C09080=1091.233,-110.223,-49.572,174.703,15.869,152.459
C09081=1091.239,-109.973,-49.581,174.704,15.869,152.459
C09082=1091.245,-109.724,-49.590,174.706,15.870,152.459
C09083=1091.251,-109.474,-49.600,174.708,15.871,152.459
C09084=1091.257,-109.224,-49.610,174.709,15.871,152.458
C09085=1091.263,-108.974,-49.619,174.711,15.872,152.458
C09086=1091.270,-108.724,-49.629,174.713,15.872,152.458
C09087=1091.275,-108.475,-49.640,174.714,15.872,152.458
C09088=1091.281,-108.225,-49.649,174.716,15.873,152.457
C09089=1091.288,-107.975,-49.659,174.717,15.874,152.457
C09090=1091.294,-107.726,-49.668,174.719,15.874,152.457
C09091=1091.300,-107.476,-49.678,174.720,15.875,152.457
C09092=1091.306,-107.226,-49.687,174.722,15.875,152.457
C09093=1091.312,-106.976,-49.697,174.723,15.875,152.456
C09094=1091.318,-106.727,-49.708,174.725,15.877,152.456
C09095=1091.324,-106.477,-49.717,174.727,15.877,152.456
C09096=1091.330,-106.227,-49.727,174.729,15.878,152.456
C09097=1091.337,-105.977,-49.737,174.730,15.878,152.456
C09098=1091.343,-105.727,-49.746,174.732,15.879,152.455
C09099=1091.349,-105.478,-49.757,174.733,15.880,152.455
C09100=1091.355,-105.228,-49.767,174.735,15.880,152.455
C09101=1091.361,-104.978,-49.776,174.736,15.880,152.455
C09102=1091.367,-104.729,-49.786,174.738,15.881,152.454
C09103=1091.372,-104.478,-49.796,174.739,15.882,152.454
C09104=1091.379,-104.229,-49.806,174.741,15.882,152.454
C09105=1091.385,-103.980,-49.816,174.743,15.883,152.454
C09106=1091.391,-103.730,-49.825,174.745,15.884,152.454
C09107=1091.397,-103.480,-49.835,174.746,15.884,152.453
C09108=1091.403,-103.230,-49.846,174.748,15.885,152.453
C09109=1091.409,-102.981,-49.855,174.750,15.885,152.453
C09110=1091.416,-102.731,-49.865,174.750,15.886,152.453
C09111=1091.422,-102.481,-49.874,174.752,15.887,152.453
C09112=1091.427,-102.232,-49.885,174.754,15.887,152.452
C09113=1091.434,-101.982,-49.895,174.756,15.888,152.452
C09114=1091.440,-101.732,-49.904,174.757,15.889,152.452
C09115=1091.446,-101.482,-49.915,174.759,15.889,152.452
C09116=1091.452,-101.233,-49.925,174.761,15.890,152.451
C09117=1091.458,-100.983,-49.934,174.762,15.890,152.451
C09118=1091.464,-100.733,-49.944,174.763,15.891,152.451
C09119=1091.470,-100.484,-49.955,174.765,15.892,152.451
C09120=1091.476,-100.234,-49.964,174.767,15.892,152.451
C09121=1091.482,-99.984,-49.974,174.768,15.893,152.451
C09122=1091.488,-99.734,-49.985,174.770,15.894,152.450
C09123=1091.495,-99.484,-49.995,174.772,15.894,152.450
C09124=1091.501,-99.234,-50.004,174.773,15.895,152.450
C09125=1091.507,-98.985,-50.015,174.775,15.895,152.450
C09126=1091.513,-98.735,-50.025,174.776,15.896,152.449
C09127=1091.519,-98.486,-50.035,174.778,15.897,152.449
C09128=1091.525,-98.236,-50.045,174.780,15.898,152.449
C09129=1091.531,-97.986,-50.055,174.781,15.898,152.449
C09130=1091.537,-97.737,-50.065,174.783,15.899,152.449
C09131=1091.543,-97.487,-50.075,174.785,15.900,152.448
C09132=1091.550,-97.211,-50.086,174.786,15.900,152.448
C09133=1091.556,-96.936,-50.098,174.788,15.901,152.448
C09134=1091.563,-96.661,-50.109,174.790,15.902,152.448
C09135=1091.570,-96.385,-50.119,174.791,15.902,152.448
C09136=1091.575,-96.135,-50.130,174.793,15.903,152.447
C09137=1091.582,-95.886,-50.140,174.795,15.904,152.447
C09138=1091.587,-95.636,-50.150,174.796,15.905,152.447
C09139=1091.593,-95.387,-50.160,174.798,15.906,152.447
C09140=1091.600,-95.136,-50.171,174.799,15.906,152.447
C09141=1091.606,-94.887,-50.181,174.801,15.907,152.446
C09142=1091.611,-94.637,-50.191,174.803,15.908,152.446
C09143=1091.618,-94.387,-50.201,174.805,15.908,152.446
C09144=1091.623,-94.138,-50.212,174.805,15.909,152.446
C09145=1091.629,-93.888,-50.221,174.807,15.910,152.446
C09146=1091.635,-93.638,-50.232,174.809,15.911,152.446
C09147=1091.641,-93.388,-50.242,174.811,15.911,152.445
C09148=1091.647,-93.139,-50.253,174.812,15.911,152.445
C09149=1091.653,-92.889,-50.262,174.813,15.913,152.445
C09150=1091.659,-92.640,-50.273,174.815,15.913,152.445
C09151=1091.665,-92.390,-50.283,174.817,15.914,152.445
C09152=1091.671,-92.140,-50.294,174.819,15.915,152.444
C09153=1091.678,-91.890,-50.303,174.820,15.916,152.444
C09154=1091.683,-91.640,-50.314,174.822,15.916,152.444
C09155=1091.690,-91.391,-50.324,174.824,15.917,152.444
C09156=1091.695,-91.141,-50.335,174.825,15.918,152.444
C09157=1091.701,-90.892,-50.346,174.826,15.918,152.443
C09158=1091.707,-90.642,-50.355,174.828,15.919,152.443
C09159=1091.713,-90.392,-50.366,174.830,15.920,152.443
C09160=1091.719,-90.143,-50.376,174.831,15.921,152.443
C09161=1091.726,-89.892,-50.387,174.833,15.922,152.443
C09162=1091.732,-89.643,-50.396,174.834,15.922,152.442
C09163=1091.737,-89.393,-50.407,174.836,15.923,152.442
C09164=1091.744,-89.144,-50.418,174.838,15.924,152.442
C09165=1091.749,-88.894,-50.428,174.839,15.925,152.442
C09166=1091.755,-88.644,-50.439,174.841,15.925,152.442
C09167=1091.761,-88.394,-50.448,174.842,15.926,152.442
C09168=1091.768,-88.144,-50.460,174.844,15.927,152.441
C09169=1091.774,-87.895,-50.470,174.846,15.928,152.441
C09170=1091.780,-87.645,-50.480,174.848,15.928,152.441
C09171=1091.786,-87.396,-50.490,174.849,15.930,152.441
C09172=1091.791,-87.146,-50.500,174.850,15.930,152.441
C09173=1091.797,-86.896,-50.511,174.852,15.931,152.441
C09174=1091.804,-86.646,-50.522,174.854,15.931,152.440
C09175=1091.810,-86.396,-50.532,174.856,15.932,152.440
C09176=1091.816,-86.147,-50.542,174.857,15.933,152.440
C09177=1091.822,-85.898,-50.553,174.858,15.933,152.440
C09178=1091.828,-85.648,-50.563,174.860,15.934,152.440
C09179=1091.834,-85.398,-50.574,174.862,15.935,152.439
C09180=1091.840,-85.148,-50.585,174.864,15.936,152.439
C09181=1091.846,-84.898,-50.594,174.865,15.937,152.439
C09182=1091.852,-84.649,-50.605,174.866,15.937,152.439
C09183=1091.858,-84.399,-50.616,174.868,15.938,152.439
C09184=1091.865,-84.149,-50.627,174.870,15.939,152.438
C09185=1091.870,-83.899,-50.637,174.872,15.940,152.438
C09186=1091.877,-83.650,-50.647,174.873,15.941,152.438
C09187=1091.883,-83.401,-50.658,174.875,15.942,152.438
C09188=1091.889,-83.150,-50.669,174.876,15.942,152.438
C09189=1091.895,-82.901,-50.679,174.878,15.943,152.438
C09190=1091.901,-82.651,-50.690,174.879,15.944,152.437
C09191=1091.907,-82.402,-50.701,174.881,15.945,152.437
C09192=1091.914,-82.152,-50.711,174.883,15.946,152.437
C09193=1091.919,-81.902,-50.722,174.885,15.946,152.437
C09194=1091.926,-81.652,-50.732,174.886,15.947,152.437
C09195=1091.931,-81.403,-50.743,174.888,15.948,152.436
C09196=1091.938,-81.130,-50.754,174.889,15.949,152.436
C09197=1091.945,-80.856,-50.766,174.891,15.950,152.436
C09198=1091.951,-80.584,-50.778,174.893,15.951,152.436
C09199=1091.958,-80.310,-50.789,174.895,15.951,152.436
C09200=1091.964,-80.061,-50.800,174.896,15.952,152.436
C09201=1091.970,-79.812,-50.811,174.898,15.953,152.435
C09202=1091.976,-79.561,-50.821,174.900,15.954,152.435
C09203=1091.982,-79.311,-50.832,174.902,15.955,152.435
C09204=1091.988,-79.062,-50.843,174.903,15.956,152.435
C09205=1091.994,-78.812,-50.854,174.904,15.956,152.435
C09206=1092.001,-78.562,-50.864,174.906,15.957,152.435
C09207=1092.006,-78.313,-50.875,174.908,15.958,152.434
C09208=1092.012,-78.063,-50.886,174.909,15.959,152.434
C09209=1092.018,-77.813,-50.896,174.911,15.960,152.434
C09210=1092.024,-77.563,-50.908,174.913,15.961,152.434
C09211=1092.030,-77.314,-50.918,174.915,15.962,152.434
C09212=1092.036,-77.064,-50.929,174.915,15.963,152.434
C09213=1092.042,-76.815,-50.940,174.917,15.963,152.433
C09214=1092.048,-76.565,-50.951,174.919,15.964,152.433
C09215=1092.054,-76.315,-50.962,174.921,15.965,152.433
C09216=1092.060,-76.066,-50.973,174.922,15.966,152.433
C09217=1092.065,-75.816,-50.983,174.924,15.967,152.433
C09218=1092.072,-75.566,-50.993,174.926,15.968,152.433
C09219=1092.078,-75.316,-51.004,174.927,15.969,152.432
C09220=1092.084,-75.067,-51.015,174.929,15.969,152.432
C09221=1092.090,-74.817,-51.026,174.930,15.970,152.432
C09222=1092.096,-74.567,-51.037,174.932,15.972,152.432
C09223=1092.101,-74.318,-51.048,174.934,15.972,152.432
C09224=1092.107,-74.068,-51.059,174.935,15.973,152.432
C09225=1092.114,-73.818,-51.070,174.937,15.974,152.432
C09226=1092.119,-73.568,-51.081,174.939,15.975,152.431
C09227=1092.125,-73.319,-51.092,174.940,15.976,152.431
C09228=1092.131,-73.070,-51.103,174.941,15.977,152.431
C09229=1092.137,-72.819,-51.114,174.943,15.977,152.431
C09230=1092.143,-72.570,-51.125,174.945,15.979,152.431
C09231=1092.149,-72.320,-51.136,174.946,15.980,152.431
C09232=1092.154,-72.071,-51.147,174.948,15.981,152.431
C09233=1092.161,-71.821,-51.158,174.950,15.982,152.430
C09234=1092.166,-71.571,-51.169,174.951,15.983,152.430
C09235=1092.172,-71.322,-51.180,174.953,15.984,152.430
C09236=1092.179,-71.071,-51.191,174.955,15.985,152.430
C09237=1092.184,-70.822,-51.202,174.957,15.986,152.430
C09238=1092.190,-70.572,-51.213,174.957,15.986,152.430
C09239=1092.196,-70.323,-51.224,174.959,15.987,152.429
C09240=1092.202,-70.073,-51.235,174.961,15.988,152.429
C09241=1092.208,-69.823,-51.246,174.962,15.989,152.429
C09242=1092.213,-69.574,-51.257,174.964,15.990,152.429
C09243=1092.219,-69.323,-51.269,174.966,15.991,152.429
C09244=1092.225,-69.074,-51.279,174.968,15.992,152.429
C09245=1092.231,-68.825,-51.291,174.969,15.993,152.429
C09246=1092.237,-68.575,-51.302,174.971,15.994,152.428
C09247=1092.243,-68.325,-51.313,174.973,15.995,152.428
C09248=1092.249,-68.076,-51.324,174.974,15.996,152.428
C09249=1092.254,-67.826,-51.335,174.975,15.997,152.428
C09250=1092.261,-67.576,-51.346,174.977,15.998,152.428
C09251=1092.267,-67.327,-51.357,174.979,15.999,152.428
C09252=1092.272,-67.077,-51.368,174.980,16.000,152.428
C09253=1092.278,-66.827,-51.380,174.982,16.001,152.427
C09254=1092.284,-66.578,-51.391,174.984,16.002,152.427
C09255=1092.290,-66.328,-51.403,174.985,16.003,152.427
C09256=1092.296,-66.078,-51.413,174.987,16.004,152.427
C09257=1092.302,-65.829,-51.424,174.989,16.005,152.427
C09258=1092.308,-65.578,-51.436,174.990,16.006,152.427
C09259=1092.314,-65.329,-51.446,174.992,16.007,152.426
C09260=1092.320,-65.058,-51.459,174.994,16.008,152.426
C09261=1092.327,-64.788,-51.471,174.995,16.009,152.426
C09262=1092.333,-64.517,-51.483,174.997,16.010,152.426
C09263=1092.340,-64.245,-51.495,174.999,16.011,152.426
C09264=1092.345,-63.995,-51.507,175.001,16.012,152.426
C09265=1092.351,-63.746,-51.518,175.002,16.013,152.426
C09266=1092.357,-63.496,-51.530,175.004,16.014,152.425
C09267=1092.363,-63.247,-51.541,175.005,16.015,152.425
C09268=1092.369,-62.997,-51.552,175.007,16.016,152.425
C09269=1092.376,-62.748,-51.563,175.009,16.017,152.425
C09270=1092.381,-62.498,-51.574,175.011,16.018,152.425
C09271=1092.387,-62.248,-51.586,175.012,16.019,152.425
C09272=1092.393,-61.998,-51.597,175.014,16.020,152.424
C09273=1092.399,-61.749,-51.609,175.016,16.021,152.424
C09274=1092.405,-61.499,-51.620,175.017,16.022,152.424
C09275=1092.411,-61.249,-51.631,175.018,16.023,152.424
C09276=1092.417,-61.000,-51.643,175.020,16.023,152.424
C09277=1092.422,-60.750,-51.654,175.022,16.025,152.424
C09278=1092.429,-60.500,-51.665,175.023,16.026,152.424
C09279=1092.435,-60.251,-51.677,175.025,16.027,152.424
C09280=1092.441,-60.001,-51.688,175.027,16.027,152.423
C09281=1092.447,-59.752,-51.699,175.028,16.029,152.423
C09282=1092.453,-59.502,-51.712,175.030,16.030,152.423
C09283=1092.458,-59.252,-51.723,175.032,16.030,152.423
C09284=1092.465,-59.002,-51.734,175.033,16.032,152.423
C09285=1092.471,-58.753,-51.745,175.035,16.033,152.423
C09286=1092.477,-58.503,-51.757,175.037,16.034,152.423
C09287=1092.482,-58.253,-51.768,175.038,16.035,152.422
C09288=1092.489,-58.004,-51.780,175.040,16.036,152.422
C09289=1092.495,-57.754,-51.791,175.042,16.037,152.422
C09290=1092.501,-57.504,-51.802,175.043,16.038,152.422
C09291=1092.506,-57.255,-51.814,175.045,16.039,152.422
C09292=1092.513,-57.004,-51.826,175.047,16.040,152.422
C09293=1092.519,-56.756,-51.837,175.048,16.041,152.422
C09294=1092.525,-56.505,-51.848,175.050,16.042,152.421
C09295=1092.530,-56.256,-51.861,175.052,16.043,152.421
C09296=1092.537,-56.006,-51.872,175.053,16.044,152.421
C09297=1092.542,-55.757,-51.883,175.055,16.045,152.421
C09298=1092.549,-55.507,-51.895,175.057,16.046,152.421
C09299=1092.555,-55.258,-51.906,175.059,16.047,152.421
C09300=1092.561,-55.008,-51.918,175.060,16.048,152.421
C09301=1092.566,-54.758,-51.929,175.062,16.049,152.420
C09302=1092.573,-54.509,-51.941,175.063,16.050,152.420
C09303=1092.578,-54.259,-51.952,175.065,16.051,152.420
C09304=1092.585,-54.009,-51.964,175.067,16.052,152.420
C09305=1092.590,-53.760,-51.975,175.069,16.053,152.420
C09306=1092.597,-53.510,-51.987,175.070,16.054,152.420
C09307=1092.603,-53.260,-51.999,175.072,16.055,152.419
C09308=1092.609,-53.011,-52.011,175.074,16.056,152.419
C09309=1092.615,-52.761,-52.022,175.075,16.057,152.419
C09310=1092.621,-52.512,-52.034,175.077,16.059,152.419
C09311=1092.627,-52.261,-52.045,175.078,16.059,152.419
C09312=1092.633,-52.012,-52.057,175.080,16.060,152.419
C09313=1092.639,-51.762,-52.068,175.081,16.061,152.419
C09314=1092.645,-51.512,-52.081,175.083,16.062,152.419
C09315=1092.651,-51.263,-52.092,175.085,16.063,152.418
C09316=1092.657,-51.013,-52.104,175.086,16.064,152.418
C09317=1092.663,-50.764,-52.116,175.088,16.065,152.418
C09318=1092.669,-50.514,-52.127,175.089,16.066,152.418
C09319=1092.676,-50.264,-52.139,175.091,16.067,152.418
C09320=1092.681,-50.014,-52.150,175.094,16.069,152.418
C09321=1092.687,-49.765,-52.162,175.095,16.070,152.418
C09322=1092.693,-49.516,-52.175,175.097,16.071,152.417
C09323=1092.699,-49.265,-52.186,175.099,16.072,152.417
C09324=1092.705,-48.996,-52.199,175.100,16.073,152.417
C09325=1092.711,-48.727,-52.212,175.102,16.074,152.417
C09326=1092.717,-48.457,-52.225,175.103,16.075,152.417
C09327=1092.723,-48.187,-52.237,175.105,16.076,152.417
C09328=1092.730,-47.938,-52.249,175.107,16.077,152.417
C09329=1092.735,-47.688,-52.261,175.108,16.078,152.417
C09330=1092.742,-47.438,-52.273,175.110,16.080,152.416
C09331=1092.747,-47.189,-52.285,175.112,16.081,152.416
C09332=1092.753,-46.939,-52.296,175.113,16.082,152.416
C09333=1092.759,-46.689,-52.309,175.115,16.083,152.416
C09334=1092.765,-46.440,-52.321,175.117,16.084,152.416
C09335=1092.771,-46.190,-52.332,175.118,16.085,152.416
C09336=1092.776,-45.941,-52.344,175.121,16.087,152.416
C09337=1092.783,-45.691,-52.356,175.122,16.088,152.416
C09338=1092.789,-45.441,-52.368,175.124,16.089,152.415
C09339=1092.795,-45.192,-52.380,175.126,16.090,152.415
C09340=1092.801,-44.942,-52.392,175.127,16.091,152.415
C09341=1092.806,-44.693,-52.405,175.129,16.092,152.415
C09342=1092.812,-44.442,-52.416,175.131,16.093,152.415
C09343=1092.818,-44.193,-52.428,175.132,16.094,152.415
C09344=1092.824,-43.944,-52.440,175.134,16.095,152.415
C09345=1092.830,-43.693,-52.452,175.136,16.096,152.415
C09346=1092.836,-43.444,-52.463,175.137,16.098,152.414
C09347=1092.842,-43.194,-52.476,175.139,16.099,152.414
C09348=1092.848,-42.945,-52.489,175.141,16.099,152.414
C09349=1092.854,-42.696,-52.500,175.142,16.101,152.414
C09350=1092.859,-42.445,-52.512,175.144,16.102,152.414
C09351=1092.865,-42.195,-52.525,175.145,16.103,152.414
C09352=1092.871,-41.946,-52.536,175.147,16.104,152.414
C09353=1092.877,-41.697,-52.549,175.149,16.105,152.414
C09354=1092.884,-41.447,-52.561,175.150,16.106,152.413
C09355=1092.889,-41.197,-52.572,175.152,16.107,152.413
C09356=1092.895,-40.947,-52.585,175.154,16.108,152.413
C09357=1092.901,-40.698,-52.597,175.155,16.109,152.413
C09358=1092.907,-40.448,-52.609,175.157,16.110,152.413
C09359=1092.912,-40.199,-52.621,175.159,16.112,152.413
C09360=1092.919,-39.949,-52.633,175.161,16.113,152.413
C09361=1092.924,-39.700,-52.646,175.163,16.114,152.412
C09362=1092.930,-39.449,-52.657,175.164,16.115,152.412
C09363=1092.937,-39.200,-52.669,175.166,16.116,152.412
C09364=1092.942,-38.951,-52.682,175.168,16.117,152.412
C09365=1092.949,-38.701,-52.693,175.169,16.119,152.412
C09366=1092.955,-38.451,-52.706,175.171,16.120,152.412
C09367=1092.960,-38.202,-52.718,175.173,16.121,152.412
C09368=1092.966,-37.952,-52.731,175.174,16.122,152.412
C09369=1092.972,-37.702,-52.743,175.176,16.123,152.412
C09370=1092.978,-37.453,-52.755,175.178,16.124,152.411
C09371=1092.984,-37.203,-52.767,175.179,16.125,152.411
C09372=1092.990,-36.954,-52.780,175.181,16.126,152.411
C09373=1092.995,-36.704,-52.792,175.183,16.128,152.411
C09374=1093.000,-36.454,-52.804,175.185,16.129,152.411
C09375=1093.006,-36.204,-52.817,175.186,16.130,152.411
C09376=1093.012,-35.955,-52.828,175.188,16.131,152.411
C09377=1093.018,-35.705,-52.841,175.190,16.132,152.411
C09378=1093.024,-35.455,-52.853,175.191,16.134,152.410
C09379=1093.030,-35.206,-52.865,175.193,16.135,152.410
C09380=1093.035,-34.956,-52.878,175.194,16.136,152.410
C09381=1093.041,-34.706,-52.891,175.196,16.137,152.410
C09382=1093.048,-34.457,-52.903,175.198,16.138,152.410
C09383=1093.053,-34.208,-52.915,175.200,16.139,152.410
C09384=1093.059,-33.958,-52.927,175.201,16.140,152.410
C09385=1093.065,-33.708,-52.940,175.204,16.142,152.410
C09386=1093.071,-33.458,-52.952,175.205,16.143,152.409
C09387=1093.076,-33.209,-52.965,175.207,16.144,152.409
C09388=1093.083,-32.939,-52.978,175.208,16.145,152.409
C09389=1093.090,-32.671,-52.992,175.210,16.146,152.409
C09390=1093.095,-32.401,-53.005,175.212,16.148,152.409
C09391=1093.102,-32.132,-53.019,175.214,16.149,152.409
C09392=1093.108,-31.883,-53.031,175.216,16.150,152.409
C09393=1093.114,-31.633,-53.043,175.218,16.151,152.409
C09394=1093.120,-31.383,-53.056,175.219,16.152,152.408
C09395=1093.126,-31.133,-53.068,175.221,16.153,152.408
C09396=1093.131,-30.884,-53.080,175.222,16.155,152.408
C09397=1093.137,-30.634,-53.093,175.224,16.156,152.408
C09398=1093.144,-30.385,-53.106,175.226,16.157,152.408
C09399=1093.149,-30.135,-53.119,175.228,16.159,152.408
C09400=1093.155,-29.885,-53.131,175.230,16.159,152.408
C09401=1093.161,-29.636,-53.143,175.231,16.160,152.408
C09402=1093.167,-29.386,-53.156,175.233,16.162,152.407
C09403=1093.173,-29.136,-53.168,175.235,16.163,152.407
C09404=1093.178,-28.886,-53.181,175.236,16.164,152.407
C09405=1093.185,-28.637,-53.194,175.238,16.165,152.407
C09406=1093.191,-28.388,-53.206,175.239,16.166,152.407
C09407=1093.197,-28.138,-53.218,175.241,16.167,152.407
C09408=1093.203,-27.889,-53.231,175.243,16.169,152.407
C09409=1093.208,-27.639,-53.244,175.245,16.170,152.407
C09410=1093.215,-27.389,-53.257,175.247,16.171,152.406
C09411=1093.221,-27.139,-53.269,175.249,16.172,152.406
C09412=1093.226,-26.890,-53.282,175.250,16.173,152.406
C09413=1093.232,-26.640,-53.294,175.252,16.174,152.406
C09414=1093.238,-26.391,-53.307,175.253,16.175,152.406
C09415=1093.244,-26.141,-53.320,175.255,16.177,152.406
C09416=1093.250,-25.891,-53.332,175.257,16.178,152.406
C09417=1093.254,-25.642,-53.345,175.259,16.179,152.406
C09418=1093.261,-25.393,-53.358,175.261,16.181,152.406
C09419=1093.266,-25.143,-53.371,175.262,16.182,152.405
C09420=1093.272,-24.893,-53.384,175.264,16.183,152.405
C09421=1093.278,-24.643,-53.396,175.266,16.184,152.405
C09422=1093.284,-24.394,-53.409,175.267,16.185,152.405
C09423=1093.290,-24.145,-53.422,175.269,16.186,152.405
C09424=1093.296,-23.895,-53.434,175.271,16.188,152.405
C09425=1093.302,-23.645,-53.447,175.273,16.189,152.405
C09426=1093.307,-23.395,-53.461,175.275,16.190,152.405
C09427=1093.313,-23.145,-53.473,175.276,16.191,152.404
C09428=1093.319,-22.897,-53.486,175.278,16.192,152.404
C09429=1093.325,-22.647,-53.499,175.279,16.193,152.404
C09430=1093.330,-22.397,-53.511,175.281,16.195,152.404
C09431=1093.337,-22.148,-53.524,175.283,16.196,152.404
C09432=1093.343,-21.898,-53.537,175.285,16.197,152.404
C09433=1093.348,-21.648,-53.550,175.287,16.199,152.404
C09434=1093.354,-21.398,-53.563,175.288,16.200,152.404
C09435=1093.359,-21.149,-53.576,175.290,16.200,152.403
C09436=1093.365,-20.900,-53.589,175.292,16.202,152.403
C09437=1093.371,-20.650,-53.601,175.293,16.203,152.403
C09438=1093.377,-20.400,-53.614,175.296,16.204,152.403
C09439=1093.384,-20.151,-53.627,175.297,16.206,152.403
C09440=1093.389,-19.901,-53.640,175.299,16.207,152.403
C09441=1093.395,-19.651,-53.654,175.300,16.208,152.403
C09442=1093.401,-19.402,-53.666,175.302,16.209,152.403
C09443=1093.407,-19.152,-53.679,175.304,16.210,152.403
C09444=1093.412,-18.903,-53.692,175.305,16.211,152.403
C09445=1093.417,-18.653,-53.705,175.308,16.213,152.402
C09446=1093.424,-18.404,-53.718,175.310,16.214,152.402
C09447=1093.430,-18.154,-53.731,175.311,16.215,152.402
C09448=1093.436,-17.905,-53.744,175.313,16.216,152.402
C09449=1093.442,-17.655,-53.756,175.314,16.217,152.402
C09450=1093.447,-17.405,-53.770,175.316,16.218,152.402
C09451=1093.453,-17.155,-53.783,175.318,16.220,152.402
C09452=1093.459,-16.885,-53.797,175.320,16.221,152.401
C09453=1093.465,-16.615,-53.811,175.322,16.222,152.401
C09454=1093.472,-16.345,-53.826,175.324,16.224,152.401
C09455=1093.479,-16.075,-53.840,175.326,16.225,152.401
C09456=1093.485,-15.825,-53.852,175.328,16.226,152.401
C09457=1093.491,-15.576,-53.866,175.329,16.227,152.401
C09458=1093.497,-15.326,-53.878,175.331,16.228,152.401
C09459=1093.502,-15.077,-53.892,175.333,16.230,152.401
C09460=1093.508,-14.827,-53.905,175.335,16.231,152.400
C09461=1093.514,-14.577,-53.918,175.336,16.232,152.400
C09462=1093.519,-14.329,-53.931,175.338,16.233,152.400
C09463=1093.525,-14.079,-53.944,175.340,16.235,152.400
C09464=1093.531,-13.829,-53.957,175.341,16.235,152.400
C09465=1093.537,-13.579,-53.970,175.344,16.237,152.400
C09466=1093.543,-13.330,-53.984,175.345,16.238,152.400
C09467=1093.548,-13.080,-53.998,175.347,16.239,152.400
C09468=1093.554,-12.830,-54.010,175.349,16.240,152.399
C09469=1093.560,-12.581,-54.023,175.350,16.242,152.399
C09470=1093.566,-12.331,-54.037,175.353,16.243,152.399
C09471=1093.572,-12.082,-54.050,175.354,16.244,152.399
C09472=1093.577,-11.832,-54.064,175.356,16.246,152.399
C09473=1093.583,-11.582,-54.076,175.358,16.247,152.399
C09474=1093.589,-11.333,-54.090,175.359,16.248,152.399
C09475=1093.595,-11.083,-54.103,175.361,16.249,152.399
C09476=1093.601,-10.834,-54.116,175.363,16.250,152.398
C09477=1093.606,-10.584,-54.130,175.365,16.251,152.398
C09478=1093.612,-10.335,-54.143,175.367,16.253,152.398
C09479=1093.618,-10.085,-54.157,175.368,16.254,152.398
C09480=1093.624,-9.835,-54.169,175.370,16.255,152.398
C09481=1093.630,-9.586,-54.183,175.372,16.257,152.398
C09482=1093.635,-9.336,-54.197,175.374,16.258,152.398
C09483=1093.641,-9.087,-54.209,175.375,16.259,152.398
C09484=1093.647,-8.837,-54.223,175.377,16.260,152.398
C09485=1093.653,-8.588,-54.236,175.379,16.261,152.397
C09486=1093.659,-8.338,-54.250,175.381,16.262,152.397
C09487=1093.664,-8.088,-54.263,175.383,16.264,152.397
C09488=1093.670,-7.839,-54.277,175.385,16.265,152.397
C09489=1093.676,-7.589,-54.290,175.386,16.266,152.397
C09490=1093.682,-7.340,-54.304,175.388,16.267,152.397
C09491=1093.688,-7.091,-54.317,175.390,16.269,152.397
C09492=1093.693,-6.840,-54.330,175.392,16.270,152.397
C09493=1093.699,-6.591,-54.343,175.393,16.271,152.396
C09494=1093.705,-6.342,-54.357,175.395,16.272,152.396
C09495=1093.712,-6.092,-54.371,175.397,16.273,152.396
C09496=1093.717,-5.842,-54.385,175.399,16.275,152.396
C09497=1093.723,-5.593,-54.398,175.401,16.276,152.396
C09498=1093.729,-5.343,-54.411,175.403,16.277,152.396
C09499=1093.735,-5.093,-54.424,175.404,16.278,152.396
C09500=1093.740,-4.844,-54.438,175.406,16.279,152.395
C09501=1093.746,-4.594,-54.452,175.408,16.281,152.395
C09502=1093.752,-4.345,-54.465,175.410,16.282,152.395
C09503=1093.758,-4.096,-54.479,175.412,16.283,152.395
C09504=1093.763,-3.846,-54.493,175.413,16.284,152.395
C09505=1093.770,-3.596,-54.506,175.416,16.286,152.395
C09506=1093.776,-3.346,-54.520,175.417,16.287,152.395
C09507=1093.782,-3.097,-54.533,175.419,16.288,152.394
C09508=1093.787,-2.847,-54.547,175.421,16.289,152.394
C09509=1093.793,-2.597,-54.560,175.422,16.290,152.394
C09510=1093.799,-2.348,-54.574,175.425,16.292,152.394
C09511=1093.804,-2.099,-54.588,175.426,16.293,152.394
C09512=1093.810,-1.849,-54.601,175.428,16.294,152.394
C09513=1093.815,-1.599,-54.615,175.430,16.295,152.394
C09514=1093.821,-1.350,-54.629,175.432,16.297,152.394
C09515=1093.827,-1.101,-54.642,175.434,16.298,152.394
C09516=1093.833,-0.829,-54.657,175.435,16.299,152.394
C09517=1093.839,-0.557,-54.672,175.438,16.301,152.393
C09518=1093.846,-0.285,-54.687,175.440,16.301,152.393
C09519=1093.852,-0.013,-54.702,175.442,16.303,152.393
C09520=1093.858,0.236,-54.716,175.444,16.304,152.393
C09521=1093.863,0.486,-54.730,175.445,16.305,152.393
C09522=1093.869,0.736,-54.743,175.447,16.307,152.393
C09523=1093.875,0.985,-54.757,175.448,16.308,152.393
C09524=1093.880,1.234,-54.771,175.451,16.310,152.392
C09525=1093.886,1.483,-54.785,175.452,16.311,152.392
C09526=1093.892,1.733,-54.799,175.454,16.311,152.392
C09527=1093.898,1.982,-54.812,175.456,16.312,152.392
C09528=1093.904,2.232,-54.827,175.458,16.314,152.392
C09529=1093.909,2.482,-54.840,175.460,16.315,152.392
C09530=1093.915,2.732,-54.854,175.461,16.317,152.392
C09531=1093.920,2.981,-54.868,175.463,16.318,152.392
C09532=1093.927,3.230,-54.881,175.465,16.319,152.391
C09533=1093.932,3.480,-54.895,175.467,16.321,152.391
C09534=1093.938,3.730,-54.909,175.469,16.321,152.391
C09535=1093.944,3.980,-54.923,175.471,16.322,152.391
C09536=1093.949,4.229,-54.938,175.473,16.324,152.391
C09537=1093.956,4.478,-54.951,175.475,16.325,152.391
C09538=1093.961,4.728,-54.965,175.476,16.326,152.391
C09539=1093.967,4.977,-54.979,175.478,16.328,152.391
C09540=1093.973,5.228,-54.993,175.481,16.329,152.390
C09541=1093.978,5.477,-55.007,175.482,16.330,152.390
C09542=1093.985,5.726,-55.021,175.484,16.331,152.390
C09543=1093.990,5.975,-55.035,175.485,16.332,152.390
C09544=1093.996,6.225,-55.049,175.488,16.334,152.390
C09545=1094.002,6.475,-55.063,175.490,16.335,152.390
C09546=1094.007,6.725,-55.077,175.491,16.336,152.389
C09547=1094.013,6.974,-55.091,175.493,16.337,152.389
C09548=1094.018,7.223,-55.105,175.495,16.339,152.389
C09549=1094.025,7.473,-55.119,175.497,16.340,152.389
C09550=1094.031,7.723,-55.133,175.499,16.341,152.389
C09551=1094.037,7.972,-55.147,175.500,16.342,152.389
C09552=1094.042,8.221,-55.161,175.503,16.343,152.389
C09553=1094.047,8.471,-55.175,175.504,16.345,152.389
C09554=1094.054,8.721,-55.189,175.506,16.346,152.388
C09555=1094.059,8.970,-55.204,175.508,16.346,152.388
C09556=1094.066,9.219,-55.217,175.510,16.348,152.388
C09557=1094.071,9.469,-55.231,175.512,16.349,152.388
C09558=1094.077,9.719,-55.245,175.513,16.350,152.388
C09559=1094.083,9.968,-55.260,175.516,16.352,152.388
C09560=1094.088,10.218,-55.274,175.518,16.353,152.388
C09561=1094.094,10.468,-55.288,175.519,16.354,152.387
C09562=1094.100,10.717,-55.303,175.521,16.355,152.387
C09563=1094.106,10.967,-55.316,175.524,16.356,152.387
C09564=1094.111,11.216,-55.331,175.525,16.358,152.387
C09565=1094.118,11.466,-55.345,175.527,16.359,152.387
C09566=1094.124,11.715,-55.358,175.529,16.360,152.387
C09567=1094.130,11.964,-55.373,175.531,16.361,152.386
C09568=1094.136,12.214,-55.387,175.533,16.362,152.386
C09569=1094.141,12.464,-55.401,175.534,16.363,152.386
C09570=1094.147,12.713,-55.416,175.536,16.365,152.386
C09571=1094.153,12.963,-55.430,175.539,16.366,152.386
C09572=1094.159,13.212,-55.445,175.540,16.367,152.386
C09573=1094.164,13.462,-55.458,175.542,16.368,152.386
C09574=1094.170,13.712,-55.473,175.545,16.369,152.385
C09575=1094.176,13.961,-55.487,175.546,16.370,152.385
C09576=1094.182,14.211,-55.501,175.548,16.372,152.385
C09577=1094.188,14.460,-55.516,175.549,16.373,152.385
C09578=1094.193,14.710,-55.530,175.552,16.374,152.385
C09579=1094.199,14.959,-55.544,175.554,16.375,152.385
C09580=1094.206,15.233,-55.560,175.556,16.377,152.385
C09581=1094.212,15.506,-55.576,175.558,16.378,152.384
C09582=1094.218,15.780,-55.591,175.560,16.379,152.384
C09583=1094.225,16.054,-55.607,175.562,16.380,152.384
C09584=1094.230,16.304,-55.622,175.564,16.382,152.384
C09585=1094.236,16.552,-55.637,175.566,16.383,152.384
C09586=1094.242,16.803,-55.651,175.568,16.384,152.384
C09587=1094.248,17.052,-55.665,175.570,16.385,152.383
C09588=1094.253,17.301,-55.679,175.572,16.387,152.383
C09589=1094.259,17.551,-55.694,175.574,16.388,152.383
C09590=1094.265,17.801,-55.708,175.576,16.389,152.383
C09591=1094.271,18.049,-55.723,175.577,16.390,152.383
C09592=1094.276,18.300,-55.737,175.580,16.392,152.383
C09593=1094.282,18.549,-55.752,175.581,16.392,152.383
C09594=1094.288,18.799,-55.767,175.583,16.393,152.382
C09595=1094.294,19.048,-55.781,175.585,16.395,152.382
C09596=1094.299,19.297,-55.795,175.587,16.396,152.382
C09597=1094.305,19.548,-55.810,175.589,16.397,152.382
C09598=1094.311,19.796,-55.824,175.591,16.398,152.382
C09599=1094.316,20.046,-55.839,175.593,16.399,152.382
C09600=1094.322,20.296,-55.854,175.595,16.400,152.381
C09601=1094.328,20.545,-55.868,175.596,16.402,152.381
C09602=1094.335,20.795,-55.883,175.599,16.403,152.381
C09603=1094.340,21.044,-55.897,175.601,16.404,152.381
C09604=1094.345,21.293,-55.912,175.602,16.405,152.381
C09605=1094.351,21.543,-55.927,175.605,16.407,152.381
C09606=1094.357,21.793,-55.941,175.607,16.408,152.380
C09607=1094.363,22.042,-55.956,175.608,16.409,152.380
C09608=1094.368,22.292,-55.971,175.611,16.410,152.380
C09609=1094.374,22.541,-55.985,175.613,16.411,152.380
C09610=1094.380,22.791,-56.000,175.614,16.412,152.380
C09611=1094.385,23.040,-56.015,175.617,16.414,152.380
C09612=1094.391,23.290,-56.029,175.618,16.415,152.380
C09613=1094.397,23.539,-56.044,175.620,16.416,152.379
C09614=1094.403,23.788,-56.058,175.622,16.417,152.379
C09615=1094.409,24.038,-56.074,175.624,16.418,152.379
C09616=1094.414,24.288,-56.088,175.626,16.419,152.379
C09617=1094.420,24.537,-56.103,175.628,16.421,152.379
C09618=1094.425,24.787,-56.118,175.630,16.422,152.379
C09619=1094.432,25.036,-56.133,175.632,16.423,152.378
C09620=1094.438,25.285,-56.148,175.634,16.424,152.378
C09621=1094.444,25.536,-56.162,175.636,16.425,152.378
C09622=1094.449,25.785,-56.177,175.638,16.426,152.378
C09623=1094.455,26.034,-56.191,175.639,16.428,152.378
C09624=1094.461,26.284,-56.206,175.642,16.429,152.378
C09625=1094.466,26.533,-56.222,175.644,16.430,152.378
C09626=1094.472,26.782,-56.237,175.646,16.431,152.377
C09627=1094.478,27.032,-56.250,175.648,16.432,152.377
C09628=1094.483,27.282,-56.266,175.650,16.434,152.377
C09629=1094.489,27.531,-56.281,175.652,16.434,152.377
C09630=1094.495,27.781,-56.296,175.654,16.436,152.377
C09631=1094.501,28.030,-56.311,175.656,16.437,152.376
C09632=1094.507,28.280,-56.326,175.657,16.438,152.376
C09633=1094.512,28.529,-56.341,175.660,16.440,152.376
C09634=1094.518,28.778,-56.356,175.662,16.440,152.376
C09635=1094.523,29.028,-56.370,175.663,16.441,152.376
C09636=1094.530,29.278,-56.385,175.666,16.443,152.376
C09637=1094.535,29.527,-56.400,175.668,16.444,152.375
C09638=1094.541,29.777,-56.415,175.669,16.445,152.375
C09639=1094.547,30.026,-56.430,175.672,16.446,152.375
C09640=1094.552,30.276,-56.445,175.674,16.447,152.375
C09641=1094.558,30.525,-56.460,175.675,16.448,152.375
C09642=1094.564,30.775,-56.475,175.678,16.450,152.375
C09643=1094.570,31.024,-56.490,175.679,16.451,152.375
C09644=1094.575,31.299,-56.507,175.682,16.452,152.374
C09645=1094.581,31.574,-56.523,175.684,16.453,152.374
C09646=1094.588,31.850,-56.540,175.687,16.455,152.374
C09647=1094.595,32.124,-56.557,175.688,16.456,152.374
C09648=1094.600,32.373,-56.572,175.691,16.457,152.373
C09649=1094.606,32.623,-56.587,175.692,16.458,152.373
C09650=1094.612,32.872,-56.602,175.695,16.460,152.373
C09651=1094.617,33.122,-56.617,175.697,16.460,152.373
C09652=1094.624,33.372,-56.632,175.698,16.462,152.373
C09653=1094.629,33.621,-56.648,175.701,16.463,152.373
C09654=1094.635,33.871,-56.663,175.703,16.464,152.372
C09655=1094.640,34.120,-56.678,175.705,16.465,152.372
C09656=1094.646,34.370,-56.693,175.707,16.466,152.372
C09657=1094.652,34.619,-56.708,175.709,16.467,152.372
C09658=1094.657,34.869,-56.723,175.710,16.468,152.372
C09659=1094.664,35.119,-56.738,175.713,16.469,152.371
C09660=1094.669,35.367,-56.754,175.715,16.471,152.371
C09661=1094.676,35.617,-56.769,175.717,16.471,152.371
C09662=1094.681,35.866,-56.784,175.719,16.473,152.371
C09663=1094.686,36.116,-56.800,175.721,16.474,152.371
C09664=1094.693,36.366,-56.815,175.723,16.475,152.371
C09665=1094.698,36.615,-56.830,175.725,16.476,152.370
C09666=1094.704,36.865,-56.845,175.727,16.477,152.370
C09667=1094.709,37.113,-56.861,175.730,16.478,152.370
C09668=1094.716,37.363,-56.876,175.731,16.480,152.370
C09669=1094.721,37.613,-56.891,175.733,16.480,152.370
C09670=1094.726,37.862,-56.906,175.735,16.482,152.370
C09671=1094.733,38.112,-56.921,175.737,16.483,152.369
C09672=1094.738,38.361,-56.937,175.740,16.484,152.369
C09673=1094.744,38.611,-56.953,175.742,16.485,152.369
C09674=1094.749,38.861,-56.968,175.743,16.486,152.369
C09675=1094.755,39.110,-56.983,175.746,16.488,152.368
C09676=1094.761,39.360,-56.998,175.748,16.489,152.368
C09677=1094.766,39.608,-57.014,175.749,16.489,152.368
C09678=1094.772,39.858,-57.030,175.752,16.491,152.368
C09679=1094.778,40.108,-57.045,175.754,16.492,152.368
C09680=1094.784,40.356,-57.061,175.756,16.493,152.368
C09681=1094.789,40.606,-57.076,175.758,16.494,152.367
C09682=1094.795,40.856,-57.092,175.760,16.495,152.367
C09683=1094.801,41.105,-57.106,175.762,16.497,152.367
C09684=1094.807,41.355,-57.123,175.764,16.497,152.367
C09685=1094.812,41.604,-57.138,175.766,16.498,152.367
C09686=1094.817,41.854,-57.153,175.769,16.500,152.366
C09687=1094.824,42.103,-57.169,175.770,16.501,152.366
C09688=1094.829,42.352,-57.184,175.773,16.502,152.366
C09689=1094.835,42.602,-57.200,175.775,16.503,152.366
C09690=1094.841,42.852,-57.216,175.776,16.504,152.366
C09691=1094.846,43.101,-57.231,175.779,16.505,152.365
C09692=1094.852,43.350,-57.246,175.781,16.506,152.365
C09693=1094.858,43.600,-57.262,175.783,16.507,152.365
C09694=1094.864,43.850,-57.278,175.785,16.509,152.365
C09695=1094.869,44.098,-57.294,175.787,16.509,152.365
C09696=1094.875,44.348,-57.309,175.789,16.511,152.365
C09697=1094.880,44.598,-57.325,175.791,16.512,152.364
C09698=1094.886,44.847,-57.341,175.794,16.513,152.364
C09699=1094.891,45.097,-57.356,175.796,16.514,152.364
C09700=1094.897,45.346,-57.372,175.797,16.515,152.364
C09701=1094.902,45.596,-57.388,175.800,16.517,152.364
C09702=1094.908,45.845,-57.404,175.802,16.517,152.363
C09703=1094.914,46.094,-57.419,175.804,16.519,152.363
C09704=1094.920,46.343,-57.435,175.806,16.520,152.363
C09705=1094.926,46.593,-57.450,175.808,16.520,152.363
C09706=1094.931,46.842,-57.466,175.810,16.522,152.363
C09707=1094.937,47.092,-57.482,175.812,16.523,152.362
C09708=1094.943,47.367,-57.500,175.815,16.524,152.362
C09709=1094.948,47.643,-57.517,175.817,16.526,152.362
C09710=1094.955,47.917,-57.534,175.819,16.526,152.362
C09711=1094.961,48.193,-57.552,175.822,16.528,152.361
C09712=1094.967,48.443,-57.567,175.824,16.529,152.361
C09713=1094.972,48.691,-57.583,175.826,16.530,152.361
C09714=1094.978,48.941,-57.599,175.828,16.531,152.361
C09715=1094.984,49.191,-57.615,175.830,16.532,152.361
C09716=1094.990,49.440,-57.631,175.832,16.533,152.360
C09717=1094.995,49.689,-57.647,175.834,16.534,152.360
C09718=1095.001,49.939,-57.663,175.837,16.535,152.360
C09719=1095.007,50.188,-57.678,175.839,16.536,152.360
C09720=1095.012,50.438,-57.695,175.841,16.538,152.360
C09721=1095.018,50.686,-57.711,175.843,16.539,152.359
C09722=1095.023,50.936,-57.726,175.845,16.539,152.359
C09723=1095.029,51.186,-57.742,175.847,16.541,152.359
C09724=1095.035,51.436,-57.758,175.849,16.542,152.359
C09725=1095.040,51.684,-57.774,175.852,16.543,152.358
C09726=1095.046,51.934,-57.790,175.853,16.544,152.358
C09727=1095.051,52.184,-57.806,175.856,16.545,152.358
C09728=1095.057,52.433,-57.822,175.858,16.546,152.358
C09729=1095.063,52.683,-57.839,175.860,16.547,152.358
C09730=1095.069,52.931,-57.855,175.862,16.548,152.357
C09731=1095.074,53.181,-57.870,175.864,16.549,152.357
C09732=1095.080,53.431,-57.886,175.867,16.550,152.357
C09733=1095.086,53.680,-57.903,175.869,16.551,152.357
C09734=1095.092,53.930,-57.918,175.870,16.552,152.357
C09735=1095.097,54.179,-57.934,175.873,16.553,152.356
C09736=1095.103,54.428,-57.950,175.875,16.554,152.356
C09737=1095.109,54.677,-57.967,175.878,16.555,152.356
C09738=1095.115,54.927,-57.982,175.880,16.556,152.355
C09739=1095.120,55.177,-57.999,175.882,16.558,152.355
C09740=1095.126,55.426,-58.015,175.884,16.558,152.355
C09741=1095.131,55.675,-58.031,175.886,16.559,152.355
C09742=1095.137,55.924,-58.047,175.889,16.560,152.355
C09743=1095.143,56.174,-58.063,175.890,16.561,152.354
C09744=1095.149,56.424,-58.079,175.893,16.563,152.354
C09745=1095.155,56.673,-58.095,175.895,16.563,152.354
C09746=1095.161,56.922,-58.112,175.897,16.565,152.354
C09747=1095.166,57.172,-58.128,175.899,16.565,152.353
C09748=1095.171,57.422,-58.144,175.902,16.566,152.353
C09749=1095.177,57.671,-58.160,175.904,16.567,152.353
C09750=1095.183,57.920,-58.176,175.906,16.568,152.353
C09751=1095.189,58.169,-58.192,175.908,16.570,152.353
C09752=1095.195,58.419,-58.209,175.910,16.570,152.352
C09753=1095.201,58.668,-58.225,175.913,16.572,152.352
C09754=1095.206,58.918,-58.242,175.915,16.572,152.352
C09755=1095.212,59.167,-58.258,175.917,16.573,152.351
C09756=1095.218,59.416,-58.274,175.919,16.574,152.351
C09757=1095.224,59.666,-58.291,175.921,16.575,152.351
C09758=1095.229,59.916,-58.306,175.924,16.576,152.351
C09759=1095.235,60.165,-58.322,175.925,16.577,152.351
C09760=1095.240,60.415,-58.339,175.928,16.578,152.350
C09761=1095.246,60.664,-58.355,175.930,16.579,152.350
C09762=1095.252,60.913,-58.372,175.933,16.580,152.350
C09763=1095.258,61.163,-58.388,175.935,16.581,152.350
C09764=1095.264,61.412,-58.404,175.937,16.582,152.349
C09765=1095.269,61.662,-58.421,175.939,16.583,152.349
C09766=1095.275,61.911,-58.437,175.941,16.584,152.349
C09767=1095.281,62.160,-58.454,175.944,16.585,152.348
C09768=1095.287,62.409,-58.469,175.946,16.586,152.348
C09769=1095.292,62.659,-58.486,175.948,16.587,152.348
C09770=1095.298,62.908,-58.503,175.950,16.587,152.348
C09771=1095.305,63.158,-58.520,175.953,16.589,152.347
C09772=1095.311,63.433,-58.538,175.955,16.589,152.347
C09773=1095.317,63.708,-58.556,175.958,16.591,152.347
C09774=1095.323,63.982,-58.574,175.960,16.592,152.347
C09775=1095.330,64.257,-58.591,175.963,16.592,152.346
C09776=1095.335,64.507,-58.608,175.965,16.593,152.346
C09777=1095.341,64.756,-58.625,175.967,16.594,152.346
C09778=1095.347,65.005,-58.642,175.970,16.596,152.346
C09779=1095.353,65.254,-58.658,175.971,16.596,152.345
C09780=1095.359,65.504,-58.675,175.974,16.598,152.345
C09781=1095.364,65.753,-58.691,175.976,16.598,152.345
C09782=1095.370,66.003,-58.708,175.979,16.600,152.344
C09783=1095.375,66.253,-58.725,175.981,16.600,152.344
C09784=1095.381,66.502,-58.741,175.983,16.602,152.344
C09785=1095.387,66.751,-58.758,175.985,16.602,152.344
C09786=1095.392,67.000,-58.775,175.988,16.603,152.343
C09787=1095.398,67.250,-58.791,175.990,16.604,152.343
C09788=1095.404,67.499,-58.808,175.993,16.605,152.343
C09789=1095.410,67.749,-58.824,175.994,16.606,152.343
C09790=1095.415,67.998,-58.842,175.996,16.607,152.342
C09791=1095.421,68.247,-58.858,175.999,16.608,152.342
C09792=1095.426,68.497,-58.875,176.001,16.608,152.342
C09793=1095.432,68.746,-58.891,176.004,16.609,152.341
C09794=1095.437,68.996,-58.908,176.006,16.610,152.341
C09795=1095.444,69.244,-58.925,176.008,16.611,152.341
C09796=1095.449,69.494,-58.942,176.010,16.612,152.341
C09797=1095.455,69.743,-58.958,176.013,16.613,152.340
C09798=1095.461,69.993,-58.976,176.015,16.614,152.340
C09799=1095.467,70.242,-58.992,176.018,16.615,152.340
C09800=1095.472,70.492,-59.009,176.020,16.616,152.340
C09801=1095.478,70.741,-59.025,176.022,16.617,152.339
C09802=1095.484,70.991,-59.043,176.024,16.618,152.339
C09803=1095.490,71.240,-59.059,176.027,16.619,152.339
C09804=1095.495,71.490,-59.076,176.029,16.620,152.339
C09805=1095.500,71.739,-59.093,176.031,16.621,152.338
C09806=1095.506,71.988,-59.110,176.034,16.621,152.338
C09807=1095.511,72.238,-59.127,176.036,16.622,152.338
C09808=1095.518,72.486,-59.144,176.038,16.623,152.337
C09809=1095.523,72.736,-59.160,176.041,16.624,152.337
C09810=1095.528,72.985,-59.178,176.043,16.625,152.337
C09811=1095.534,73.234,-59.194,176.045,16.626,152.337
C09812=1095.540,73.484,-59.211,176.047,16.627,152.336
C09813=1095.546,73.734,-59.229,176.050,16.628,152.336
C09814=1095.552,73.983,-59.245,176.052,16.629,152.336
C09815=1095.557,74.232,-59.263,176.055,16.630,152.335
C09816=1095.563,74.481,-59.279,176.057,16.630,152.335
C09817=1095.569,74.731,-59.297,176.060,16.632,152.335
C09818=1095.574,74.980,-59.313,176.061,16.632,152.335
C09819=1095.580,75.230,-59.330,176.064,16.634,152.334
C09820=1095.585,75.479,-59.347,176.066,16.634,152.334
C09821=1095.591,75.728,-59.364,176.068,16.634,152.334
C09822=1095.597,75.978,-59.381,176.071,16.636,152.333
C09823=1095.603,76.227,-59.398,176.073,16.636,152.333
C09824=1095.608,76.476,-59.416,176.076,16.638,152.333
C09825=1095.614,76.726,-59.432,176.077,16.638,152.333
C09826=1095.620,76.975,-59.450,176.080,16.639,152.332
C09827=1095.625,77.224,-59.467,176.082,16.640,152.332
C09828=1095.631,77.474,-59.485,176.085,16.641,152.332
C09829=1095.637,77.723,-59.501,176.087,16.642,152.331
C09830=1095.642,77.973,-59.518,176.090,16.643,152.331
C09831=1095.648,78.222,-59.536,176.092,16.643,152.331
C09832=1095.653,78.471,-59.553,176.094,16.644,152.330
C09833=1095.659,78.720,-59.570,176.096,16.645,152.330
C09834=1095.665,78.970,-59.588,176.099,16.646,152.330
C09835=1095.671,79.219,-59.605,176.102,16.647,152.330
C09836=1095.677,79.494,-59.623,176.104,16.648,152.329
C09837=1095.683,79.769,-59.642,176.107,16.649,152.329
C09838=1095.689,80.044,-59.662,176.110,16.650,152.329
C09839=1095.695,80.319,-59.680,176.112,16.651,152.328
C09840=1095.701,80.568,-59.698,176.114,16.651,152.328
C09841=1095.706,80.817,-59.715,176.117,16.653,152.328
C09842=1095.712,81.067,-59.733,176.119,16.653,152.327
C09843=1095.718,81.316,-59.750,176.122,16.655,152.327
C09844=1095.723,81.565,-59.768,176.124,16.655,152.327
C09845=1095.729,81.815,-59.784,176.127,16.656,152.326
C09846=1095.735,82.064,-59.802,176.129,16.657,152.326
C09847=1095.741,82.313,-59.820,176.131,16.658,152.326
C09848=1095.746,82.562,-59.837,176.133,16.658,152.325
C09849=1095.752,82.812,-59.854,176.136,16.659,152.325
C09850=1095.757,83.061,-59.872,176.138,16.660,152.325
C09851=1095.763,83.310,-59.889,176.141,16.661,152.325
C09852=1095.768,83.561,-59.906,176.143,16.662,152.324
C09853=1095.774,83.810,-59.924,176.146,16.663,152.324
C09854=1095.779,84.059,-59.941,176.148,16.663,152.324
C09855=1095.785,84.308,-59.959,176.150,16.664,152.323
C09856=1095.792,84.557,-59.976,176.153,16.664,152.323
C09857=1095.797,84.807,-59.993,176.155,16.666,152.323
C09858=1095.803,85.056,-60.011,176.157,16.666,152.322
C09859=1095.808,85.305,-60.028,176.160,16.667,152.322
C09860=1095.814,85.555,-60.046,176.163,16.668,152.322
C09861=1095.820,85.804,-60.064,176.165,16.669,152.321
C09862=1095.825,86.053,-60.081,176.168,16.670,152.321
C09863=1095.831,86.303,-60.099,176.170,16.671,152.321
C09864=1095.837,86.552,-60.116,176.173,16.671,152.320
C09865=1095.842,86.801,-60.134,176.175,16.672,152.320
C09866=1095.848,87.050,-60.151,176.178,16.673,152.320
C09867=1095.854,87.300,-60.169,176.179,16.674,152.319
C09868=1095.859,87.549,-60.187,176.182,16.674,152.319
C09869=1095.865,87.798,-60.204,176.184,16.675,152.319
C09870=1095.871,88.048,-60.222,176.187,16.676,152.318
C09871=1095.876,88.297,-60.240,176.189,16.676,152.318
C09872=1095.882,88.546,-60.257,176.192,16.678,152.318
C09873=1095.888,88.795,-60.275,176.194,16.678,152.317
C09874=1095.894,89.045,-60.293,176.197,16.679,152.317
C09875=1095.899,89.294,-60.311,176.199,16.679,152.317
C09876=1095.905,89.543,-60.328,176.202,16.680,152.316
C09877=1095.911,89.792,-60.346,176.205,16.681,152.316
C09878=1095.917,90.042,-60.364,176.207,16.682,152.316
C09879=1095.922,90.291,-60.382,176.210,16.683,152.315
C09880=1095.928,90.540,-60.399,176.212,16.683,152.315
C09881=1095.934,90.790,-60.417,176.214,16.684,152.315
C09882=1095.939,91.039,-60.435,176.217,16.685,152.314
C09883=1095.944,91.288,-60.453,176.219,16.686,152.314
C09884=1095.950,91.538,-60.471,176.221,16.686,152.314
C09885=1095.956,91.787,-60.488,176.224,16.687,152.313
C09886=1095.961,92.036,-60.506,176.226,16.688,152.313
C09887=1095.968,92.286,-60.524,176.229,16.689,152.313
C09888=1095.972,92.535,-60.542,176.232,16.690,152.312
C09889=1095.978,92.784,-60.559,176.234,16.690,152.312
C09890=1095.984,93.034,-60.577,176.237,16.691,152.312
C09891=1095.989,93.283,-60.595,176.239,16.692,152.311
C09892=1095.996,93.533,-60.613,176.242,16.693,152.311
C09893=1096.001,93.782,-60.632,176.244,16.693,152.310
C09894=1096.006,94.031,-60.649,176.247,16.694,152.310
C09895=1096.012,94.280,-60.667,176.249,16.694,152.310
C09896=1096.018,94.529,-60.685,176.252,16.695,152.310
C09897=1096.023,94.779,-60.703,176.254,16.696,152.309
C09898=1096.029,95.028,-60.721,176.256,16.697,152.309
C09899=1096.035,95.277,-60.739,176.259,16.698,152.308
C09900=1096.041,95.552,-60.759,176.262,16.698,152.308
C09901=1096.047,95.827,-60.779,176.265,16.699,152.308
C09902=1096.053,96.102,-60.798,176.267,16.700,152.307
C09903=1096.060,96.377,-60.818,176.270,16.701,152.307
C09904=1096.066,96.627,-60.836,176.272,16.701,152.307
C09905=1096.071,96.875,-60.855,176.275,16.702,152.306
C09906=1096.076,97.124,-60.873,176.278,16.703,152.306
C09907=1096.082,97.374,-60.891,176.280,16.703,152.305
C09908=1096.087,97.624,-60.909,176.283,16.704,152.305
C09909=1096.094,97.873,-60.928,176.285,16.705,152.305
C09910=1096.099,98.122,-60.945,176.288,16.706,152.304
C09911=1096.105,98.371,-60.963,176.290,16.706,152.304
C09912=1096.110,98.620,-60.982,176.293,16.707,152.304
C09913=1096.116,98.870,-61.000,176.296,16.708,152.303
C09914=1096.122,99.119,-61.017,176.298,16.708,152.303
C09915=1096.128,99.368,-61.037,176.301,16.709,152.302
C09916=1096.133,99.617,-61.054,176.303,16.709,152.302
C09917=1096.139,99.867,-61.072,176.306,16.710,152.302
C09918=1096.144,100.116,-61.091,176.308,16.710,152.301
C09919=1096.150,100.366,-61.109,176.311,16.711,152.301
C09920=1096.156,100.615,-61.127,176.313,16.712,152.301
C09921=1096.162,100.864,-61.146,176.316,16.713,152.300
C09922=1096.167,101.113,-61.163,176.319,16.714,152.300
C09923=1096.174,101.362,-61.182,176.321,16.714,152.299
C09924=1096.178,101.612,-61.200,176.324,16.715,152.299
C09925=1096.185,101.861,-61.219,176.326,16.715,152.299
C09926=1096.190,102.110,-61.237,176.329,16.716,152.298
C09927=1096.196,102.360,-61.255,176.332,16.717,152.298
C09928=1096.201,102.609,-61.274,176.334,16.717,152.297
C09929=1096.207,102.858,-61.292,176.337,16.718,152.297
C09930=1096.212,103.107,-61.311,176.339,16.718,152.297
C09931=1096.218,103.357,-61.329,176.342,16.719,152.296
C09932=1096.223,103.606,-61.347,176.344,16.719,152.296
C09933=1096.229,103.855,-61.365,176.347,16.721,152.296
C09934=1096.234,104.104,-61.384,176.350,16.722,152.295
C09935=1096.241,104.354,-61.402,176.352,16.722,152.295
C09936=1096.246,104.602,-61.421,176.355,16.723,152.294
C09937=1096.251,104.853,-61.440,176.357,16.723,152.294
C09938=1096.257,105.102,-61.458,176.360,16.724,152.294
C09939=1096.263,105.350,-61.477,176.363,16.725,152.293
C09940=1096.269,105.600,-61.495,176.365,16.725,152.293
C09941=1096.274,105.849,-61.514,176.368,16.726,152.293
C09942=1096.280,106.099,-61.532,176.370,16.726,152.292
C09943=1096.285,106.347,-61.551,176.373,16.727,152.292
C09944=1096.291,106.596,-61.569,176.375,16.727,152.291
C09945=1096.297,106.847,-61.588,176.378,16.728,152.291
C09946=1096.302,107.095,-61.607,176.381,16.729,152.290
C09947=1096.308,107.345,-61.625,176.383,16.729,152.290
C09948=1096.313,107.594,-61.644,176.386,16.730,152.290
C09949=1096.319,107.843,-61.662,176.388,16.730,152.289
C09950=1096.325,108.093,-61.681,176.391,16.731,152.289
C09951=1096.330,108.342,-61.700,176.394,16.732,152.289
C09952=1096.336,108.591,-61.718,176.397,16.732,152.288
C09953=1096.341,108.840,-61.736,176.400,16.733,152.288
C09954=1096.348,109.089,-61.755,176.402,16.733,152.287
C09955=1096.353,109.339,-61.774,176.405,16.734,152.287
C09956=1096.358,109.587,-61.793,176.408,16.735,152.286
C09957=1096.364,109.837,-61.811,176.410,16.735,152.286
C09958=1096.370,110.087,-61.830,176.413,16.736,152.286
C09959=1096.376,110.335,-61.849,176.415,16.736,152.285
C09960=1096.382,110.584,-61.868,176.418,16.737,152.285
C09961=1096.387,110.834,-61.886,176.421,16.738,152.284
C09962=1096.393,111.083,-61.905,176.423,16.738,152.284
C09963=1096.399,111.332,-61.924,176.426,16.739,152.284
C09964=1096.404,111.608,-61.945,176.429,16.739,152.283
C09965=1096.411,111.882,-61.966,176.432,16.740,152.283
C09966=1096.417,112.157,-61.987,176.435,16.740,152.282
C09967=1096.424,112.432,-62.007,176.438,16.741,152.282
C09968=1096.429,112.681,-62.026,176.441,16.742,152.281
C09969=1096.435,112.931,-62.045,176.444,16.742,152.281
C09970=1096.440,113.180,-62.064,176.446,16.743,152.281
C09971=1096.446,113.429,-62.082,176.449,16.743,152.280
C09972=1096.452,113.679,-62.101,176.451,16.744,152.280
C09973=1096.457,113.927,-62.120,176.454,16.744,152.279
C09974=1096.463,114.177,-62.139,176.457,16.745,152.279
C09975=1096.469,114.426,-62.158,176.459,16.745,152.278
C09976=1096.475,114.675,-62.177,176.462,16.746,152.278
C09977=1096.480,114.924,-62.196,176.464,16.746,152.277
C09978=1096.486,115.174,-62.215,176.467,16.747,152.277
C09979=1096.491,115.423,-62.235,176.470,16.748,152.277
C09980=1096.496,115.672,-62.254,176.473,16.748,152.276
C09981=1096.502,115.921,-62.273,176.476,16.749,152.276
C09982=1096.508,116.171,-62.292,176.479,16.749,152.275
C09983=1096.513,116.419,-62.311,176.481,16.750,152.275
C09984=1096.518,116.669,-62.330,176.484,16.750,152.275
C09985=1096.524,116.918,-62.349,176.486,16.751,152.274
C09986=1096.529,117.167,-62.368,176.489,16.751,152.274
C09987=1096.535,117.416,-62.388,176.492,16.752,152.273
C09988=1096.541,117.665,-62.406,176.494,16.752,152.273
C09989=1096.546,117.914,-62.425,176.497,16.753,152.272
C09990=1096.552,118.164,-62.444,176.500,16.754,152.272
C09991=1096.558,118.413,-62.464,176.502,16.754,152.272
C09992=1096.563,118.663,-62.483,176.505,16.755,152.271
C09993=1096.569,118.911,-62.502,176.508,16.755,152.271
C09994=1096.574,119.161,-62.521,176.511,16.755,152.270
C09995=1096.580,119.410,-62.540,176.514,16.756,152.270
C09996=1096.586,119.660,-62.559,176.516,16.756,152.269
//INST
///DATE 2021/06/17 10:53
///ATTR SC,RW,RJ
////FRAME ROBOT
///GROUP1 RB1
NOP
MOVL C00000 V=800.0 PL=0
MOVL C00001 V=800.0 PL=0
MOVL C00002 V=800.0 PL=0
MOVL C00003 V=800.0 PL=0
MOVL C00004 V=800.0 PL=0
MOVL C00005 V=800.0 PL=0
MOVL C00006 V=800.0 PL=0
MOVL C00007 V=800.0 PL=0
MOVL C00008 V=800.0 PL=0
MOVL C00009 V=800.0 PL=0
MOVL C00010 V=800.0 PL=0
MOVL C00011 V=800.0 PL=0
MOVL C00012 V=800.0 PL=0
MOVL C00013 V=800.0 PL=0
MOVL C00014 V=800.0 PL=0
MOVL C00015 V=800.0 PL=0
MOVL C00016 V=800.0 PL=0
MOVL C00017 V=800.0 PL=0
MOVL C00018 V=800.0 PL=0
MOVL C00019 V=800.0 PL=0
MOVL C00020 V=800.0 PL=0
MOVL C00021 V=800.0 PL=0
MOVL C00022 V=800.0 PL=0
MOVL C00023 V=800.0 PL=0
MOVL C00024 V=800.0 PL=0
MOVL C00025 V=800.0 PL=0
MOVL C00026 V=800.0 PL=0
MOVL C00027 V=800.0 PL=0
MOVL C00028 V=800.0 PL=0
MOVL C00029 V=800.0 PL=0
MOVL C00030 V=800.0 PL=0
MOVL C00031 V=800.0 PL=0
MOVL C00032 V=800.0 PL=0
MOVL C00033 V=800.0 PL=0
MOVL C00034 V=800.0 PL=0
MOVL C00035 V=800.0 PL=0
MOVL C00036 V=800.0 PL=0
MOVL C00037 V=800.0 PL=0
MOVL C00038 V=800.0 PL=0
MOVL C00039 V=800.0 PL=0
MOVL C00040 V=800.0 PL=0
MOVL C00041 V=800.0 PL=0
MOVL C00042 V=800.0 PL=0
MOVL C00043 V=800.0 PL=0
MOVL C00044 V=800.0 PL=0
MOVL C00045 V=800.0 PL=0
MOVL C00046 V=800.0 PL=0
MOVL C00047 V=800.0 PL=0
MOVL C00048 V=800.0 PL=0
MOVL C00049 V=800.0 PL=0
MOVL C00050 V=800.0 PL=0
MOVL C00051 V=800.0 PL=0
MOVL C00052 V=800.0 PL=0
MOVL C00053 V=800.0 PL=0
MOVL C00054 V=800.0 PL=0
MOVL C00055 V=800.0 PL=0
MOVL C00056 V=800.0 PL=0
MOVL C00057 V=800.0 PL=0
MOVL C00058 V=800.0 PL=0
MOVL C00059 V=800.0 PL=0
MOVL C00060 V=800.0 PL=0
MOVL C00061 V=800.0 PL=0
MOVL C00062 V=800.0 PL=0
MOVL C00063 V=800.0 PL=0
MOVL C00064 V=800.0 PL=0
MOVL C00065 V=800.0 PL=0
MOVL C00066 V=800.0 PL=0
MOVL C00067 V=800.0 PL=0
MOVL C00068 V=800.0 PL=0
MOVL C00069 V=800.0 PL=0
MOVL C00070 V=800.0 PL=0
MOVL C00071 V=800.0 PL=0
MOVL C00072 V=800.0 PL=0
MOVL C00073 V=800.0 PL=0
MOVL C00074 V=800.0 PL=0
MOVL C00075 V=800.0 PL=0
MOVL C00076 V=800.0 PL=0
MOVL C00077 V=800.0 PL=0
MOVL C00078 V=800.0 PL=0
MOVL C00079 V=800.0 PL=0
MOVL C00080 V=800.0 PL=0
MOVL C00081 V=800.0 PL=0
MOVL C00082 V=800.0 PL=0
MOVL C00083 V=800.0 PL=0
MOVL C00084 V=800.0 PL=0
MOVL C00085 V=800.0 PL=0
MOVL C00086 V=800.0 PL=0
MOVL C00087 V=800.0 PL=0
MOVL C00088 V=800.0 PL=0
MOVL C00089 V=800.0 PL=0
MOVL C00090 V=800.0 PL=0
MOVL C00091 V=800.0 PL=0
MOVL C00092 V=800.0 PL=0
MOVL C00093 V=800.0 PL=0
MOVL C00094 V=800.0 PL=0
MOVL C00095 V=800.0 PL=0
MOVL C00096 V=800.0 PL=0
MOVL C00097 V=800.0 PL=0
MOVL C00098 V=800.0 PL=0
MOVL C00099 V=800.0 PL=0
MOVL C00100 V=800.0 PL=0
MOVL C00101 V=800.0 PL=0
MOVL C00102 V=800.0 PL=0
MOVL C00103 V=800.0 PL=0
MOVL C00104 V=800.0 PL=0
MOVL C00105 V=800.0 PL=0
MOVL C00106 V=800.0 PL=0
MOVL C00107 V=800.0 PL=0
MOVL C00108 V=800.0 PL=0
MOVL C00109 V=800.0 PL=0
MOVL C00110 V=800.0 PL=0
MOVL C00111 V=800.0 PL=0
MOVL C00112 V=800.0 PL=0
MOVL C00113 V=800.0 PL=0
MOVL C00114 V=800.0 PL=0
MOVL C00115 V=800.0 PL=0
MOVL C00116 V=800.0 PL=0
MOVL C00117 V=800.0 PL=0
MOVL C00118 V=800.0 PL=0
MOVL C00119 V=800.0 PL=0
MOVL C00120 V=800.0 PL=0
MOVL C00121 V=800.0 PL=0
MOVL C00122 V=800.0 PL=0
MOVL C00123 V=800.0 PL=0
MOVL C00124 V=800.0 PL=0
MOVL C00125 V=800.0 PL=0
MOVL C00126 V=800.0 PL=0
MOVL C00127 V=800.0 PL=0
MOVL C00128 V=800.0 PL=0
MOVL C00129 V=800.0 PL=0
MOVL C00130 V=800.0 PL=0
MOVL C00131 V=800.0 PL=0
MOVL C00132 V=800.0 PL=0
MOVL C00133 V=800.0 PL=0
MOVL C00134 V=800.0 PL=0
MOVL C00135 V=800.0 PL=0
MOVL C00136 V=800.0 PL=0
MOVL C00137 V=800.0 PL=0
MOVL C00138 V=800.0 PL=0
MOVL C00139 V=800.0 PL=0
MOVL C00140 V=800.0 PL=0
MOVL C00141 V=800.0 PL=0
MOVL C00142 V=800.0 PL=0
MOVL C00143 V=800.0 PL=0
MOVL C00144 V=800.0 PL=0
MOVL C00145 V=800.0 PL=0
MOVL C00146 V=800.0 PL=0
MOVL C00147 V=800.0 PL=0
MOVL C00148 V=800.0 PL=0
MOVL C00149 V=800.0 PL=0
MOVL C00150 V=800.0 PL=0
MOVL C00151 V=800.0 PL=0
MOVL C00152 V=800.0 PL=0
MOVL C00153 V=800.0 PL=0
MOVL C00154 V=800.0 PL=0
MOVL C00155 V=800.0 PL=0
MOVL C00156 V=800.0 PL=0
MOVL C00157 V=800.0 PL=0
MOVL C00158 V=800.0 PL=0
MOVL C00159 V=800.0 PL=0
MOVL C00160 V=800.0 PL=0
MOVL C00161 V=800.0 PL=0
MOVL C00162 V=800.0 PL=0
MOVL C00163 V=800.0 PL=0
MOVL C00164 V=800.0 PL=0
MOVL C00165 V=800.0 PL=0
MOVL C00166 V=800.0 PL=0
MOVL C00167 V=800.0 PL=0
MOVL C00168 V=800.0 PL=0
MOVL C00169 V=800.0 PL=0
MOVL C00170 V=800.0 PL=0
MOVL C00171 V=800.0 PL=0
MOVL C00172 V=800.0 PL=0
MOVL C00173 V=800.0 PL=0
MOVL C00174 V=800.0 PL=0
MOVL C00175 V=800.0 PL=0
MOVL C00176 V=800.0 PL=0
MOVL C00177 V=800.0 PL=0
MOVL C00178 V=800.0 PL=0
MOVL C00179 V=800.0 PL=0
MOVL C00180 V=800.0 PL=0
MOVL C00181 V=800.0 PL=0
MOVL C00182 V=800.0 PL=0
MOVL C00183 V=800.0 PL=0
MOVL C00184 V=800.0 PL=0
MOVL C00185 V=800.0 PL=0
MOVL C00186 V=800.0 PL=0
MOVL C00187 V=800.0 PL=0
MOVL C00188 V=800.0 PL=0
MOVL C00189 V=800.0 PL=0
MOVL C00190 V=800.0 PL=0
MOVL C00191 V=800.0 PL=0
MOVL C00192 V=800.0 PL=0
MOVL C00193 V=800.0 PL=0
MOVL C00194 V=800.0 PL=0
MOVL C00195 V=800.0 PL=0
MOVL C00196 V=800.0 PL=0
MOVL C00197 V=800.0 PL=0
MOVL C00198 V=800.0 PL=0
MOVL C00199 V=800.0 PL=0
MOVL C00200 V=800.0 PL=0
MOVL C00201 V=800.0 PL=0
MOVL C00202 V=800.0 PL=0
MOVL C00203 V=800.0 PL=0
MOVL C00204 V=800.0 PL=0
MOVL C00205 V=800.0 PL=0
MOVL C00206 V=800.0 PL=0
MOVL C00207 V=800.0 PL=0
MOVL C00208 V=800.0 PL=0
MOVL C00209 V=800.0 PL=0
MOVL C00210 V=800.0 PL=0
MOVL C00211 V=800.0 PL=0
MOVL C00212 V=800.0 PL=0
MOVL C00213 V=800.0 PL=0
MOVL C00214 V=800.0 PL=0
MOVL C00215 V=800.0 PL=0
MOVL C00216 V=800.0 PL=0
MOVL C00217 V=800.0 PL=0
MOVL C00218 V=800.0 PL=0
MOVL C00219 V=800.0 PL=0
MOVL C00220 V=800.0 PL=0
MOVL C00221 V=800.0 PL=0
MOVL C00222 V=800.0 PL=0
MOVL C00223 V=800.0 PL=0
MOVL C00224 V=800.0 PL=0
MOVL C00225 V=800.0 PL=0
MOVL C00226 V=800.0 PL=0
MOVL C00227 V=800.0 PL=0
MOVL C00228 V=800.0 PL=0
MOVL C00229 V=800.0 PL=0
MOVL C00230 V=800.0 PL=0
MOVL C00231 V=800.0 PL=0
MOVL C00232 V=800.0 PL=0
MOVL C00233 V=800.0 PL=0
MOVL C00234 V=800.0 PL=0
MOVL C00235 V=800.0 PL=0
MOVL C00236 V=800.0 PL=0
MOVL C00237 V=800.0 PL=0
MOVL C00238 V=800.0 PL=0
MOVL C00239 V=800.0 PL=0
MOVL C00240 V=800.0 PL=0
MOVL C00241 V=800.0 PL=0
MOVL C00242 V=800.0 PL=0
MOVL C00243 V=800.0 PL=0
MOVL C00244 V=800.0 PL=0
MOVL C00245 V=800.0 PL=0
MOVL C00246 V=800.0 PL=0
MOVL C00247 V=800.0 PL=0
MOVL C00248 V=800.0 PL=0
MOVL C00249 V=800.0 PL=0
MOVL C00250 V=800.0 PL=0
MOVL C00251 V=800.0 PL=0
MOVL C00252 V=800.0 PL=0
MOVL C00253 V=800.0 PL=0
MOVL C00254 V=800.0 PL=0
MOVL C00255 V=800.0 PL=0
MOVL C00256 V=800.0 PL=0
MOVL C00257 V=800.0 PL=0
MOVL C00258 V=800.0 PL=0
MOVL C00259 V=800.0 PL=0
MOVL C00260 V=800.0 PL=0
MOVL C00261 V=800.0 PL=0
MOVL C00262 V=800.0 PL=0
MOVL C00263 V=800.0 PL=0
MOVL C00264 V=800.0 PL=0
MOVL C00265 V=800.0 PL=0
MOVL C00266 V=800.0 PL=0
MOVL C00267 V=800.0 PL=0
MOVL C00268 V=800.0 PL=0
MOVL C00269 V=800.0 PL=0
MOVL C00270 V=800.0 PL=0
MOVL C00271 V=800.0 PL=0
MOVL C00272 V=800.0 PL=0
MOVL C00273 V=800.0 PL=0
MOVL C00274 V=800.0 PL=0
MOVL C00275 V=800.0 PL=0
MOVL C00276 V=800.0 PL=0
MOVL C00277 V=800.0 PL=0
MOVL C00278 V=800.0 PL=0
MOVL C00279 V=800.0 PL=0
MOVL C00280 V=800.0 PL=0
MOVL C00281 V=800.0 PL=0
MOVL C00282 V=800.0 PL=0
MOVL C00283 V=800.0 PL=0
MOVL C00284 V=800.0 PL=0
MOVL C00285 V=800.0 PL=0
MOVL C00286 V=800.0 PL=0
MOVL C00287 V=800.0 PL=0
MOVL C00288 V=800.0 PL=0
MOVL C00289 V=800.0 PL=0
MOVL C00290 V=800.0 PL=0
MOVL C00291 V=800.0 PL=0
MOVL C00292 V=800.0 PL=0
MOVL C00293 V=800.0 PL=0
MOVL C00294 V=800.0 PL=0
MOVL C00295 V=800.0 PL=0
MOVL C00296 V=800.0 PL=0
MOVL C00297 V=800.0 PL=0
MOVL C00298 V=800.0 PL=0
MOVL C00299 V=800.0 PL=0
MOVL C00300 V=800.0 PL=0
MOVL C00301 V=800.0 PL=0
MOVL C00302 V=800.0 PL=0
MOVL C00303 V=800.0 PL=0
MOVL C00304 V=800.0 PL=0
MOVL C00305 V=800.0 PL=0
MOVL C00306 V=800.0 PL=0
MOVL C00307 V=800.0 PL=0
MOVL C00308 V=800.0 PL=0
MOVL C00309 V=800.0 PL=0
MOVL C00310 V=800.0 PL=0
MOVL C00311 V=800.0 PL=0
MOVL C00312 V=800.0 PL=0
MOVL C00313 V=800.0 PL=0
MOVL C00314 V=800.0 PL=0
MOVL C00315 V=800.0 PL=0
MOVL C00316 V=800.0 PL=0
MOVL C00317 V=800.0 PL=0
MOVL C00318 V=800.0 PL=0
MOVL C00319 V=800.0 PL=0
MOVL C00320 V=800.0 PL=0
MOVL C00321 V=800.0 PL=0
MOVL C00322 V=800.0 PL=0
MOVL C00323 V=800.0 PL=0
MOVL C00324 V=800.0 PL=0
MOVL C00325 V=800.0 PL=0
MOVL C00326 V=800.0 PL=0
MOVL C00327 V=800.0 PL=0
MOVL C00328 V=800.0 PL=0
MOVL C00329 V=800.0 PL=0
MOVL C00330 V=800.0 PL=0
MOVL C00331 V=800.0 PL=0
MOVL C00332 V=800.0 PL=0
MOVL C00333 V=800.0 PL=0
MOVL C00334 V=800.0 PL=0
MOVL C00335 V=800.0 PL=0
MOVL C00336 V=800.0 PL=0
MOVL C00337 V=800.0 PL=0
MOVL C00338 V=800.0 PL=0
MOVL C00339 V=800.0 PL=0
MOVL C00340 V=800.0 PL=0
MOVL C00341 V=800.0 PL=0
MOVL C00342 V=800.0 PL=0
MOVL C00343 V=800.0 PL=0
MOVL C00344 V=800.0 PL=0
MOVL C00345 V=800.0 PL=0
MOVL C00346 V=800.0 PL=0
MOVL C00347 V=800.0 PL=0
MOVL C00348 V=800.0 PL=0
MOVL C00349 V=800.0 PL=0
MOVL C00350 V=800.0 PL=0
MOVL C00351 V=800.0 PL=0
MOVL C00352 V=800.0 PL=0
MOVL C00353 V=800.0 PL=0
MOVL C00354 V=800.0 PL=0
MOVL C00355 V=800.0 PL=0
MOVL C00356 V=800.0 PL=0
MOVL C00357 V=800.0 PL=0
MOVL C00358 V=800.0 PL=0
MOVL C00359 V=800.0 PL=0
MOVL C00360 V=800.0 PL=0
MOVL C00361 V=800.0 PL=0
MOVL C00362 V=800.0 PL=0
MOVL C00363 V=800.0 PL=0
MOVL C00364 V=800.0 PL=0
MOVL C00365 V=800.0 PL=0
MOVL C00366 V=800.0 PL=0
MOVL C00367 V=800.0 PL=0
MOVL C00368 V=800.0 PL=0
MOVL C00369 V=800.0 PL=0
MOVL C00370 V=800.0 PL=0
MOVL C00371 V=800.0 PL=0
MOVL C00372 V=800.0 PL=0
MOVL C00373 V=800.0 PL=0
MOVL C00374 V=800.0 PL=0
MOVL C00375 V=800.0 PL=0
MOVL C00376 V=800.0 PL=0
MOVL C00377 V=800.0 PL=0
MOVL C00378 V=800.0 PL=0
MOVL C00379 V=800.0 PL=0
MOVL C00380 V=800.0 PL=0
MOVL C00381 V=800.0 PL=0
MOVL C00382 V=800.0 PL=0
MOVL C00383 V=800.0 PL=0
MOVL C00384 V=800.0 PL=0
MOVL C00385 V=800.0 PL=0
MOVL C00386 V=800.0 PL=0
MOVL C00387 V=800.0 PL=0
MOVL C00388 V=800.0 PL=0
MOVL C00389 V=800.0 PL=0
MOVL C00390 V=800.0 PL=0
MOVL C00391 V=800.0 PL=0
MOVL C00392 V=800.0 PL=0
MOVL C00393 V=800.0 PL=0
MOVL C00394 V=800.0 PL=0
MOVL C00395 V=800.0 PL=0
MOVL C00396 V=800.0 PL=0
MOVL C00397 V=800.0 PL=0
MOVL C00398 V=800.0 PL=0
MOVL C00399 V=800.0 PL=0
MOVL C00400 V=800.0 PL=0
MOVL C00401 V=800.0 PL=0
MOVL C00402 V=800.0 PL=0
MOVL C00403 V=800.0 PL=0
MOVL C00404 V=800.0 PL=0
MOVL C00405 V=800.0 PL=0
MOVL C00406 V=800.0 PL=0
MOVL C00407 V=800.0 PL=0
MOVL C00408 V=800.0 PL=0
MOVL C00409 V=800.0 PL=0
MOVL C00410 V=800.0 PL=0
MOVL C00411 V=800.0 PL=0
MOVL C00412 V=800.0 PL=0
MOVL C00413 V=800.0 PL=0
MOVL C00414 V=800.0 PL=0
MOVL C00415 V=800.0 PL=0
MOVL C00416 V=800.0 PL=0
MOVL C00417 V=800.0 PL=0
MOVL C00418 V=800.0 PL=0
MOVL C00419 V=800.0 PL=0
MOVL C00420 V=800.0 PL=0
MOVL C00421 V=800.0 PL=0
MOVL C00422 V=800.0 PL=0
MOVL C00423 V=800.0 PL=0
MOVL C00424 V=800.0 PL=0
MOVL C00425 V=800.0 PL=0
MOVL C00426 V=800.0 PL=0
MOVL C00427 V=800.0 PL=0
MOVL C00428 V=800.0 PL=0
MOVL C00429 V=800.0 PL=0
MOVL C00430 V=800.0 PL=0
MOVL C00431 V=800.0 PL=0
MOVL C00432 V=800.0 PL=0
MOVL C00433 V=800.0 PL=0
MOVL C00434 V=800.0 PL=0
MOVL C00435 V=800.0 PL=0
MOVL C00436 V=800.0 PL=0
MOVL C00437 V=800.0 PL=0
MOVL C00438 V=800.0 PL=0
MOVL C00439 V=800.0 PL=0
MOVL C00440 V=800.0 PL=0
MOVL C00441 V=800.0 PL=0
MOVL C00442 V=800.0 PL=0
MOVL C00443 V=800.0 PL=0
MOVL C00444 V=800.0 PL=0
MOVL C00445 V=800.0 PL=0
MOVL C00446 V=800.0 PL=0
MOVL C00447 V=800.0 PL=0
MOVL C00448 V=800.0 PL=0
MOVL C00449 V=800.0 PL=0
MOVL C00450 V=800.0 PL=0
MOVL C00451 V=800.0 PL=0
MOVL C00452 V=800.0 PL=0
MOVL C00453 V=800.0 PL=0
MOVL C00454 V=800.0 PL=0
MOVL C00455 V=800.0 PL=0
MOVL C00456 V=800.0 PL=0
MOVL C00457 V=800.0 PL=0
MOVL C00458 V=800.0 PL=0
MOVL C00459 V=800.0 PL=0
MOVL C00460 V=800.0 PL=0
MOVL C00461 V=800.0 PL=0
MOVL C00462 V=800.0 PL=0
MOVL C00463 V=800.0 PL=0
MOVL C00464 V=800.0 PL=0
MOVL C00465 V=800.0 PL=0
MOVL C00466 V=800.0 PL=0
MOVL C00467 V=800.0 PL=0
MOVL C00468 V=800.0 PL=0
MOVL C00469 V=800.0 PL=0
MOVL C00470 V=800.0 PL=0
MOVL C00471 V=800.0 PL=0
MOVL C00472 V=800.0 PL=0
MOVL C00473 V=800.0 PL=0
MOVL C00474 V=800.0 PL=0
MOVL C00475 V=800.0 PL=0
MOVL C00476 V=800.0 PL=0
MOVL C00477 V=800.0 PL=0
MOVL C00478 V=800.0 PL=0
MOVL C00479 V=800.0 PL=0
MOVL C00480 V=800.0 PL=0
MOVL C00481 V=800.0 PL=0
MOVL C00482 V=800.0 PL=0
MOVL C00483 V=800.0 PL=0
MOVL C00484 V=800.0 PL=0
MOVL C00485 V=800.0 PL=0
MOVL C00486 V=800.0 PL=0
MOVL C00487 V=800.0 PL=0
MOVL C00488 V=800.0 PL=0
MOVL C00489 V=800.0 PL=0
MOVL C00490 V=800.0 PL=0
MOVL C00491 V=800.0 PL=0
MOVL C00492 V=800.0 PL=0
MOVL C00493 V=800.0 PL=0
MOVL C00494 V=800.0 PL=0
MOVL C00495 V=800.0 PL=0
MOVL C00496 V=800.0 PL=0
MOVL C00497 V=800.0 PL=0
MOVL C00498 V=800.0 PL=0
MOVL C00499 V=800.0 PL=0
MOVL C00500 V=800.0 PL=0
MOVL C00501 V=800.0 PL=0
MOVL C00502 V=800.0 PL=0
MOVL C00503 V=800.0 PL=0
MOVL C00504 V=800.0 PL=0
MOVL C00505 V=800.0 PL=0
MOVL C00506 V=800.0 PL=0
MOVL C00507 V=800.0 PL=0
MOVL C00508 V=800.0 PL=0
MOVL C00509 V=800.0 PL=0
MOVL C00510 V=800.0 PL=0
MOVL C00511 V=800.0 PL=0
MOVL C00512 V=800.0 PL=0
MOVL C00513 V=800.0 PL=0
MOVL C00514 V=800.0 PL=0
MOVL C00515 V=800.0 PL=0
MOVL C00516 V=800.0 PL=0
MOVL C00517 V=800.0 PL=0
MOVL C00518 V=800.0 PL=0
MOVL C00519 V=800.0 PL=0
MOVL C00520 V=800.0 PL=0
MOVL C00521 V=800.0 PL=0
MOVL C00522 V=800.0 PL=0
MOVL C00523 V=800.0 PL=0
MOVL C00524 V=800.0 PL=0
MOVL C00525 V=800.0 PL=0
MOVL C00526 V=800.0 PL=0
MOVL C00527 V=800.0 PL=0
MOVL C00528 V=800.0 PL=0
MOVL C00529 V=800.0 PL=0
MOVL C00530 V=800.0 PL=0
MOVL C00531 V=800.0 PL=0
MOVL C00532 V=800.0 PL=0
MOVL C00533 V=800.0 PL=0
MOVL C00534 V=800.0 PL=0
MOVL C00535 V=800.0 PL=0
MOVL C00536 V=800.0 PL=0
MOVL C00537 V=800.0 PL=0
MOVL C00538 V=800.0 PL=0
MOVL C00539 V=800.0 PL=0
MOVL C00540 V=800.0 PL=0
MOVL C00541 V=800.0 PL=0
MOVL C00542 V=800.0 PL=0
MOVL C00543 V=800.0 PL=0
MOVL C00544 V=800.0 PL=0
MOVL C00545 V=800.0 PL=0
MOVL C00546 V=800.0 PL=0
MOVL C00547 V=800.0 PL=0
MOVL C00548 V=800.0 PL=0
MOVL C00549 V=800.0 PL=0
MOVL C00550 V=800.0 PL=0
MOVL C00551 V=800.0 PL=0
MOVL C00552 V=800.0 PL=0
MOVL C00553 V=800.0 PL=0
MOVL C00554 V=800.0 PL=0
MOVL C00555 V=800.0 PL=0
MOVL C00556 V=800.0 PL=0
MOVL C00557 V=800.0 PL=0
MOVL C00558 V=800.0 PL=0
MOVL C00559 V=800.0 PL=0
MOVL C00560 V=800.0 PL=0
MOVL C00561 V=800.0 PL=0
MOVL C00562 V=800.0 PL=0
MOVL C00563 V=800.0 PL=0
MOVL C00564 V=800.0 PL=0
MOVL C00565 V=800.0 PL=0
MOVL C00566 V=800.0 PL=0
MOVL C00567 V=800.0 PL=0
MOVL C00568 V=800.0 PL=0
MOVL C00569 V=800.0 PL=0
MOVL C00570 V=800.0 PL=0
MOVL C00571 V=800.0 PL=0
MOVL C00572 V=800.0 PL=0
MOVL C00573 V=800.0 PL=0
MOVL C00574 V=800.0 PL=0
MOVL C00575 V=800.0 PL=0
MOVL C00576 V=800.0 PL=0
MOVL C00577 V=800.0 PL=0
MOVL C00578 V=800.0 PL=0
MOVL C00579 V=800.0 PL=0
MOVL C00580 V=800.0 PL=0
MOVL C00581 V=800.0 PL=0
MOVL C00582 V=800.0 PL=0
MOVL C00583 V=800.0 PL=0
MOVL C00584 V=800.0 PL=0
MOVL C00585 V=800.0 PL=0
MOVL C00586 V=800.0 PL=0
MOVL C00587 V=800.0 PL=0
MOVL C00588 V=800.0 PL=0
MOVL C00589 V=800.0 PL=0
MOVL C00590 V=800.0 PL=0
MOVL C00591 V=800.0 PL=0
MOVL C00592 V=800.0 PL=0
MOVL C00593 V=800.0 PL=0
MOVL C00594 V=800.0 PL=0
MOVL C00595 V=800.0 PL=0
MOVL C00596 V=800.0 PL=0
MOVL C00597 V=800.0 PL=0
MOVL C00598 V=800.0 PL=0
MOVL C00599 V=800.0 PL=0
MOVL C00600 V=800.0 PL=0
MOVL C00601 V=800.0 PL=0
MOVL C00602 V=800.0 PL=0
MOVL C00603 V=800.0 PL=0
MOVL C00604 V=800.0 PL=0
MOVL C00605 V=800.0 PL=0
MOVL C00606 V=800.0 PL=0
MOVL C00607 V=800.0 PL=0
MOVL C00608 V=800.0 PL=0
MOVL C00609 V=800.0 PL=0
MOVL C00610 V=800.0 PL=0
MOVL C00611 V=800.0 PL=0
MOVL C00612 V=800.0 PL=0
MOVL C00613 V=800.0 PL=0
MOVL C00614 V=800.0 PL=0
MOVL C00615 V=800.0 PL=0
MOVL C00616 V=800.0 PL=0
MOVL C00617 V=800.0 PL=0
MOVL C00618 V=800.0 PL=0
MOVL C00619 V=800.0 PL=0
MOVL C00620 V=800.0 PL=0
MOVL C00621 V=800.0 PL=0
MOVL C00622 V=800.0 PL=0
MOVL C00623 V=800.0 PL=0
MOVL C00624 V=800.0 PL=0
MOVL C00625 V=800.0 PL=0
MOVL C00626 V=800.0 PL=0
MOVL C00627 V=800.0 PL=0
MOVL C00628 V=800.0 PL=0
MOVL C00629 V=800.0 PL=0
MOVL C00630 V=800.0 PL=0
MOVL C00631 V=800.0 PL=0
MOVL C00632 V=800.0 PL=0
MOVL C00633 V=800.0 PL=0
MOVL C00634 V=800.0 PL=0
MOVL C00635 V=800.0 PL=0
MOVL C00636 V=800.0 PL=0
MOVL C00637 V=800.0 PL=0
MOVL C00638 V=800.0 PL=0
MOVL C00639 V=800.0 PL=0
MOVL C00640 V=800.0 PL=0
MOVL C00641 V=800.0 PL=0
MOVL C00642 V=800.0 PL=0
MOVL C00643 V=800.0 PL=0
MOVL C00644 V=800.0 PL=0
MOVL C00645 V=800.0 PL=0
MOVL C00646 V=800.0 PL=0
MOVL C00647 V=800.0 PL=0
MOVL C00648 V=800.0 PL=0
MOVL C00649 V=800.0 PL=0
MOVL C00650 V=800.0 PL=0
MOVL C00651 V=800.0 PL=0
MOVL C00652 V=800.0 PL=0
MOVL C00653 V=800.0 PL=0
MOVL C00654 V=800.0 PL=0
MOVL C00655 V=800.0 PL=0
MOVL C00656 V=800.0 PL=0
MOVL C00657 V=800.0 PL=0
MOVL C00658 V=800.0 PL=0
MOVL C00659 V=800.0 PL=0
MOVL C00660 V=800.0 PL=0
MOVL C00661 V=800.0 PL=0
MOVL C00662 V=800.0 PL=0
MOVL C00663 V=800.0 PL=0
MOVL C00664 V=800.0 PL=0
MOVL C00665 V=800.0 PL=0
MOVL C00666 V=800.0 PL=0
MOVL C00667 V=800.0 PL=0
MOVL C00668 V=800.0 PL=0
MOVL C00669 V=800.0 PL=0
MOVL C00670 V=800.0 PL=0
MOVL C00671 V=800.0 PL=0
MOVL C00672 V=800.0 PL=0
MOVL C00673 V=800.0 PL=0
MOVL C00674 V=800.0 PL=0
MOVL C00675 V=800.0 PL=0
MOVL C00676 V=800.0 PL=0
MOVL C00677 V=800.0 PL=0
MOVL C00678 V=800.0 PL=0
MOVL C00679 V=800.0 PL=0
MOVL C00680 V=800.0 PL=0
MOVL C00681 V=800.0 PL=0
MOVL C00682 V=800.0 PL=0
MOVL C00683 V=800.0 PL=0
MOVL C00684 V=800.0 PL=0
MOVL C00685 V=800.0 PL=0
MOVL C00686 V=800.0 PL=0
MOVL C00687 V=800.0 PL=0
MOVL C00688 V=800.0 PL=0
MOVL C00689 V=800.0 PL=0
MOVL C00690 V=800.0 PL=0
MOVL C00691 V=800.0 PL=0
MOVL C00692 V=800.0 PL=0
MOVL C00693 V=800.0 PL=0
MOVL C00694 V=800.0 PL=0
MOVL C00695 V=800.0 PL=0
MOVL C00696 V=800.0 PL=0
MOVL C00697 V=800.0 PL=0
MOVL C00698 V=800.0 PL=0
MOVL C00699 V=800.0 PL=0
MOVL C00700 V=800.0 PL=0
MOVL C00701 V=800.0 PL=0
MOVL C00702 V=800.0 PL=0
MOVL C00703 V=800.0 PL=0
MOVL C00704 V=800.0 PL=0
MOVL C00705 V=800.0 PL=0
MOVL C00706 V=800.0 PL=0
MOVL C00707 V=800.0 PL=0
MOVL C00708 V=800.0 PL=0
MOVL C00709 V=800.0 PL=0
MOVL C00710 V=800.0 PL=0
MOVL C00711 V=800.0 PL=0
MOVL C00712 V=800.0 PL=0
MOVL C00713 V=800.0 PL=0
MOVL C00714 V=800.0 PL=0
MOVL C00715 V=800.0 PL=0
MOVL C00716 V=800.0 PL=0
MOVL C00717 V=800.0 PL=0
MOVL C00718 V=800.0 PL=0
MOVL C00719 V=800.0 PL=0
MOVL C00720 V=800.0 PL=0
MOVL C00721 V=800.0 PL=0
MOVL C00722 V=800.0 PL=0
MOVL C00723 V=800.0 PL=0
MOVL C00724 V=800.0 PL=0
MOVL C00725 V=800.0 PL=0
MOVL C00726 V=800.0 PL=0
MOVL C00727 V=800.0 PL=0
MOVL C00728 V=800.0 PL=0
MOVL C00729 V=800.0 PL=0
MOVL C00730 V=800.0 PL=0
MOVL C00731 V=800.0 PL=0
MOVL C00732 V=800.0 PL=0
MOVL C00733 V=800.0 PL=0
MOVL C00734 V=800.0 PL=0
MOVL C00735 V=800.0 PL=0
MOVL C00736 V=800.0 PL=0
MOVL C00737 V=800.0 PL=0
MOVL C00738 V=800.0 PL=0
MOVL C00739 V=800.0 PL=0
MOVL C00740 V=800.0 PL=0
MOVL C00741 V=800.0 PL=0
MOVL C00742 V=800.0 PL=0
MOVL C00743 V=800.0 PL=0
MOVL C00744 V=800.0 PL=0
MOVL C00745 V=800.0 PL=0
MOVL C00746 V=800.0 PL=0
MOVL C00747 V=800.0 PL=0
MOVL C00748 V=800.0 PL=0
MOVL C00749 V=800.0 PL=0
MOVL C00750 V=800.0 PL=0
MOVL C00751 V=800.0 PL=0
MOVL C00752 V=800.0 PL=0
MOVL C00753 V=800.0 PL=0
MOVL C00754 V=800.0 PL=0
MOVL C00755 V=800.0 PL=0
MOVL C00756 V=800.0 PL=0
MOVL C00757 V=800.0 PL=0
MOVL C00758 V=800.0 PL=0
MOVL C00759 V=800.0 PL=0
MOVL C00760 V=800.0 PL=0
MOVL C00761 V=800.0 PL=0
MOVL C00762 V=800.0 PL=0
MOVL C00763 V=800.0 PL=0
MOVL C00764 V=800.0 PL=0
MOVL C00765 V=800.0 PL=0
MOVL C00766 V=800.0 PL=0
MOVL C00767 V=800.0 PL=0
MOVL C00768 V=800.0 PL=0
MOVL C00769 V=800.0 PL=0
MOVL C00770 V=800.0 PL=0
MOVL C00771 V=800.0 PL=0
MOVL C00772 V=800.0 PL=0
MOVL C00773 V=800.0 PL=0
MOVL C00774 V=800.0 PL=0
MOVL C00775 V=800.0 PL=0
MOVL C00776 V=800.0 PL=0
MOVL C00777 V=800.0 PL=0
MOVL C00778 V=800.0 PL=0
MOVL C00779 V=800.0 PL=0
MOVL C00780 V=800.0 PL=0
MOVL C00781 V=800.0 PL=0
MOVL C00782 V=800.0 PL=0
MOVL C00783 V=800.0 PL=0
MOVL C00784 V=800.0 PL=0
MOVL C00785 V=800.0 PL=0
MOVL C00786 V=800.0 PL=0
MOVL C00787 V=800.0 PL=0
MOVL C00788 V=800.0 PL=0
MOVL C00789 V=800.0 PL=0
MOVL C00790 V=800.0 PL=0
MOVL C00791 V=800.0 PL=0
MOVL C00792 V=800.0 PL=0
MOVL C00793 V=800.0 PL=0
MOVL C00794 V=800.0 PL=0
MOVL C00795 V=800.0 PL=0
MOVL C00796 V=800.0 PL=0
MOVL C00797 V=800.0 PL=0
MOVL C00798 V=800.0 PL=0
MOVL C00799 V=800.0 PL=0
MOVL C00800 V=800.0 PL=0
MOVL C00801 V=800.0 PL=0
MOVL C00802 V=800.0 PL=0
MOVL C00803 V=800.0 PL=0
MOVL C00804 V=800.0 PL=0
MOVL C00805 V=800.0 PL=0
MOVL C00806 V=800.0 PL=0
MOVL C00807 V=800.0 PL=0
MOVL C00808 V=800.0 PL=0
MOVL C00809 V=800.0 PL=0
MOVL C00810 V=800.0 PL=0
MOVL C00811 V=800.0 PL=0
MOVL C00812 V=800.0 PL=0
MOVL C00813 V=800.0 PL=0
MOVL C00814 V=800.0 PL=0
MOVL C00815 V=800.0 PL=0
MOVL C00816 V=800.0 PL=0
MOVL C00817 V=800.0 PL=0
MOVL C00818 V=800.0 PL=0
MOVL C00819 V=800.0 PL=0
MOVL C00820 V=800.0 PL=0
MOVL C00821 V=800.0 PL=0
MOVL C00822 V=800.0 PL=0
MOVL C00823 V=800.0 PL=0
MOVL C00824 V=800.0 PL=0
MOVL C00825 V=800.0 PL=0
MOVL C00826 V=800.0 PL=0
MOVL C00827 V=800.0 PL=0
MOVL C00828 V=800.0 PL=0
MOVL C00829 V=800.0 PL=0
MOVL C00830 V=800.0 PL=0
MOVL C00831 V=800.0 PL=0
MOVL C00832 V=800.0 PL=0
MOVL C00833 V=800.0 PL=0
MOVL C00834 V=800.0 PL=0
MOVL C00835 V=800.0 PL=0
MOVL C00836 V=800.0 PL=0
MOVL C00837 V=800.0 PL=0
MOVL C00838 V=800.0 PL=0
MOVL C00839 V=800.0 PL=0
MOVL C00840 V=800.0 PL=0
MOVL C00841 V=800.0 PL=0
MOVL C00842 V=800.0 PL=0
MOVL C00843 V=800.0 PL=0
MOVL C00844 V=800.0 PL=0
MOVL C00845 V=800.0 PL=0
MOVL C00846 V=800.0 PL=0
MOVL C00847 V=800.0 PL=0
MOVL C00848 V=800.0 PL=0
MOVL C00849 V=800.0 PL=0
MOVL C00850 V=800.0 PL=0
MOVL C00851 V=800.0 PL=0
MOVL C00852 V=800.0 PL=0
MOVL C00853 V=800.0 PL=0
MOVL C00854 V=800.0 PL=0
MOVL C00855 V=800.0 PL=0
MOVL C00856 V=800.0 PL=0
MOVL C00857 V=800.0 PL=0
MOVL C00858 V=800.0 PL=0
MOVL C00859 V=800.0 PL=0
MOVL C00860 V=800.0 PL=0
MOVL C00861 V=800.0 PL=0
MOVL C00862 V=800.0 PL=0
MOVL C00863 V=800.0 PL=0
MOVL C00864 V=800.0 PL=0
MOVL C00865 V=800.0 PL=0
MOVL C00866 V=800.0 PL=0
MOVL C00867 V=800.0 PL=0
MOVL C00868 V=800.0 PL=0
MOVL C00869 V=800.0 PL=0
MOVL C00870 V=800.0 PL=0
MOVL C00871 V=800.0 PL=0
MOVL C00872 V=800.0 PL=0
MOVL C00873 V=800.0 PL=0
MOVL C00874 V=800.0 PL=0
MOVL C00875 V=800.0 PL=0
MOVL C00876 V=800.0 PL=0
MOVL C00877 V=800.0 PL=0
MOVL C00878 V=800.0 PL=0
MOVL C00879 V=800.0 PL=0
MOVL C00880 V=800.0 PL=0
MOVL C00881 V=800.0 PL=0
MOVL C00882 V=800.0 PL=0
MOVL C00883 V=800.0 PL=0
MOVL C00884 V=800.0 PL=0
MOVL C00885 V=800.0 PL=0
MOVL C00886 V=800.0 PL=0
MOVL C00887 V=800.0 PL=0
MOVL C00888 V=800.0 PL=0
MOVL C00889 V=800.0 PL=0
MOVL C00890 V=800.0 PL=0
MOVL C00891 V=800.0 PL=0
MOVL C00892 V=800.0 PL=0
MOVL C00893 V=800.0 PL=0
MOVL C00894 V=800.0 PL=0
MOVL C00895 V=800.0 PL=0
MOVL C00896 V=800.0 PL=0
MOVL C00897 V=800.0 PL=0
MOVL C00898 V=800.0 PL=0
MOVL C00899 V=800.0 PL=0
MOVL C00900 V=800.0 PL=0
MOVL C00901 V=800.0 PL=0
MOVL C00902 V=800.0 PL=0
MOVL C00903 V=800.0 PL=0
MOVL C00904 V=800.0 PL=0
MOVL C00905 V=800.0 PL=0
MOVL C00906 V=800.0 PL=0
MOVL C00907 V=800.0 PL=0
MOVL C00908 V=800.0 PL=0
MOVL C00909 V=800.0 PL=0
MOVL C00910 V=800.0 PL=0
MOVL C00911 V=800.0 PL=0
MOVL C00912 V=800.0 PL=0
MOVL C00913 V=800.0 PL=0
MOVL C00914 V=800.0 PL=0
MOVL C00915 V=800.0 PL=0
MOVL C00916 V=800.0 PL=0
MOVL C00917 V=800.0 PL=0
MOVL C00918 V=800.0 PL=0
MOVL C00919 V=800.0 PL=0
MOVL C00920 V=800.0 PL=0
MOVL C00921 V=800.0 PL=0
MOVL C00922 V=800.0 PL=0
MOVL C00923 V=800.0 PL=0
MOVL C00924 V=800.0 PL=0
MOVL C00925 V=800.0 PL=0
MOVL C00926 V=800.0 PL=0
MOVL C00927 V=800.0 PL=0
MOVL C00928 V=800.0 PL=0
MOVL C00929 V=800.0 PL=0
MOVL C00930 V=800.0 PL=0
MOVL C00931 V=800.0 PL=0
MOVL C00932 V=800.0 PL=0
MOVL C00933 V=800.0 PL=0
MOVL C00934 V=800.0 PL=0
MOVL C00935 V=800.0 PL=0
MOVL C00936 V=800.0 PL=0
MOVL C00937 V=800.0 PL=0
MOVL C00938 V=800.0 PL=0
MOVL C00939 V=800.0 PL=0
MOVL C00940 V=800.0 PL=0
MOVL C00941 V=800.0 PL=0
MOVL C00942 V=800.0 PL=0
MOVL C00943 V=800.0 PL=0
MOVL C00944 V=800.0 PL=0
MOVL C00945 V=800.0 PL=0
MOVL C00946 V=800.0 PL=0
MOVL C00947 V=800.0 PL=0
MOVL C00948 V=800.0 PL=0
MOVL C00949 V=800.0 PL=0
MOVL C00950 V=800.0 PL=0
MOVL C00951 V=800.0 PL=0
MOVL C00952 V=800.0 PL=0
MOVL C00953 V=800.0 PL=0
MOVL C00954 V=800.0 PL=0
MOVL C00955 V=800.0 PL=0
MOVL C00956 V=800.0 PL=0
MOVL C00957 V=800.0 PL=0
MOVL C00958 V=800.0 PL=0
MOVL C00959 V=800.0 PL=0
MOVL C00960 V=800.0 PL=0
MOVL C00961 V=800.0 PL=0
MOVL C00962 V=800.0 PL=0
MOVL C00963 V=800.0 PL=0
MOVL C00964 V=800.0 PL=0
MOVL C00965 V=800.0 PL=0
MOVL C00966 V=800.0 PL=0
MOVL C00967 V=800.0 PL=0
MOVL C00968 V=800.0 PL=0
MOVL C00969 V=800.0 PL=0
MOVL C00970 V=800.0 PL=0
MOVL C00971 V=800.0 PL=0
MOVL C00972 V=800.0 PL=0
MOVL C00973 V=800.0 PL=0
MOVL C00974 V=800.0 PL=0
MOVL C00975 V=800.0 PL=0
MOVL C00976 V=800.0 PL=0
MOVL C00977 V=800.0 PL=0
MOVL C00978 V=800.0 PL=0
MOVL C00979 V=800.0 PL=0
MOVL C00980 V=800.0 PL=0
MOVL C00981 V=800.0 PL=0
MOVL C00982 V=800.0 PL=0
MOVL C00983 V=800.0 PL=0
MOVL C00984 V=800.0 PL=0
MOVL C00985 V=800.0 PL=0
MOVL C00986 V=800.0 PL=0
MOVL C00987 V=800.0 PL=0
MOVL C00988 V=800.0 PL=0
MOVL C00989 V=800.0 PL=0
MOVL C00990 V=800.0 PL=0
MOVL C00991 V=800.0 PL=0
MOVL C00992 V=800.0 PL=0
MOVL C00993 V=800.0 PL=0
MOVL C00994 V=800.0 PL=0
MOVL C00995 V=800.0 PL=0
MOVL C00996 V=800.0 PL=0
MOVL C00997 V=800.0 PL=0
MOVL C00998 V=800.0 PL=0
MOVL C00999 V=800.0 PL=0
MOVL C01000 V=800.0 PL=0
MOVL C01001 V=800.0 PL=0
MOVL C01002 V=800.0 PL=0
MOVL C01003 V=800.0 PL=0
MOVL C01004 V=800.0 PL=0
MOVL C01005 V=800.0 PL=0
MOVL C01006 V=800.0 PL=0
MOVL C01007 V=800.0 PL=0
MOVL C01008 V=800.0 PL=0
MOVL C01009 V=800.0 PL=0
MOVL C01010 V=800.0 PL=0
MOVL C01011 V=800.0 PL=0
MOVL C01012 V=800.0 PL=0
MOVL C01013 V=800.0 PL=0
MOVL C01014 V=800.0 PL=0
MOVL C01015 V=800.0 PL=0
MOVL C01016 V=800.0 PL=0
MOVL C01017 V=800.0 PL=0
MOVL C01018 V=800.0 PL=0
MOVL C01019 V=800.0 PL=0
MOVL C01020 V=800.0 PL=0
MOVL C01021 V=800.0 PL=0
MOVL C01022 V=800.0 PL=0
MOVL C01023 V=800.0 PL=0
MOVL C01024 V=800.0 PL=0
MOVL C01025 V=800.0 PL=0
MOVL C01026 V=800.0 PL=0
MOVL C01027 V=800.0 PL=0
MOVL C01028 V=800.0 PL=0
MOVL C01029 V=800.0 PL=0
MOVL C01030 V=800.0 PL=0
MOVL C01031 V=800.0 PL=0
MOVL C01032 V=800.0 PL=0
MOVL C01033 V=800.0 PL=0
MOVL C01034 V=800.0 PL=0
MOVL C01035 V=800.0 PL=0
MOVL C01036 V=800.0 PL=0
MOVL C01037 V=800.0 PL=0
MOVL C01038 V=800.0 PL=0
MOVL C01039 V=800.0 PL=0
MOVL C01040 V=800.0 PL=0
MOVL C01041 V=800.0 PL=0
MOVL C01042 V=800.0 PL=0
MOVL C01043 V=800.0 PL=0
MOVL C01044 V=800.0 PL=0
MOVL C01045 V=800.0 PL=0
MOVL C01046 V=800.0 PL=0
MOVL C01047 V=800.0 PL=0
MOVL C01048 V=800.0 PL=0
MOVL C01049 V=800.0 PL=0
MOVL C01050 V=800.0 PL=0
MOVL C01051 V=800.0 PL=0
MOVL C01052 V=800.0 PL=0
MOVL C01053 V=800.0 PL=0
MOVL C01054 V=800.0 PL=0
MOVL C01055 V=800.0 PL=0
MOVL C01056 V=800.0 PL=0
MOVL C01057 V=800.0 PL=0
MOVL C01058 V=800.0 PL=0
MOVL C01059 V=800.0 PL=0
MOVL C01060 V=800.0 PL=0
MOVL C01061 V=800.0 PL=0
MOVL C01062 V=800.0 PL=0
MOVL C01063 V=800.0 PL=0
MOVL C01064 V=800.0 PL=0
MOVL C01065 V=800.0 PL=0
MOVL C01066 V=800.0 PL=0
MOVL C01067 V=800.0 PL=0
MOVL C01068 V=800.0 PL=0
MOVL C01069 V=800.0 PL=0
MOVL C01070 V=800.0 PL=0
MOVL C01071 V=800.0 PL=0
MOVL C01072 V=800.0 PL=0
MOVL C01073 V=800.0 PL=0
MOVL C01074 V=800.0 PL=0
MOVL C01075 V=800.0 PL=0
MOVL C01076 V=800.0 PL=0
MOVL C01077 V=800.0 PL=0
MOVL C01078 V=800.0 PL=0
MOVL C01079 V=800.0 PL=0
MOVL C01080 V=800.0 PL=0
MOVL C01081 V=800.0 PL=0
MOVL C01082 V=800.0 PL=0
MOVL C01083 V=800.0 PL=0
MOVL C01084 V=800.0 PL=0
MOVL C01085 V=800.0 PL=0
MOVL C01086 V=800.0 PL=0
MOVL C01087 V=800.0 PL=0
MOVL C01088 V=800.0 PL=0
MOVL C01089 V=800.0 PL=0
MOVL C01090 V=800.0 PL=0
MOVL C01091 V=800.0 PL=0
MOVL C01092 V=800.0 PL=0
MOVL C01093 V=800.0 PL=0
MOVL C01094 V=800.0 PL=0
MOVL C01095 V=800.0 PL=0
MOVL C01096 V=800.0 PL=0
MOVL C01097 V=800.0 PL=0
MOVL C01098 V=800.0 PL=0
MOVL C01099 V=800.0 PL=0
MOVL C01100 V=800.0 PL=0
MOVL C01101 V=800.0 PL=0
MOVL C01102 V=800.0 PL=0
MOVL C01103 V=800.0 PL=0
MOVL C01104 V=800.0 PL=0
MOVL C01105 V=800.0 PL=0
MOVL C01106 V=800.0 PL=0
MOVL C01107 V=800.0 PL=0
MOVL C01108 V=800.0 PL=0
MOVL C01109 V=800.0 PL=0
MOVL C01110 V=800.0 PL=0
MOVL C01111 V=800.0 PL=0
MOVL C01112 V=800.0 PL=0
MOVL C01113 V=800.0 PL=0
MOVL C01114 V=800.0 PL=0
MOVL C01115 V=800.0 PL=0
MOVL C01116 V=800.0 PL=0
MOVL C01117 V=800.0 PL=0
MOVL C01118 V=800.0 PL=0
MOVL C01119 V=800.0 PL=0
MOVL C01120 V=800.0 PL=0
MOVL C01121 V=800.0 PL=0
MOVL C01122 V=800.0 PL=0
MOVL C01123 V=800.0 PL=0
MOVL C01124 V=800.0 PL=0
MOVL C01125 V=800.0 PL=0
MOVL C01126 V=800.0 PL=0
MOVL C01127 V=800.0 PL=0
MOVL C01128 V=800.0 PL=0
MOVL C01129 V=800.0 PL=0
MOVL C01130 V=800.0 PL=0
MOVL C01131 V=800.0 PL=0
MOVL C01132 V=800.0 PL=0
MOVL C01133 V=800.0 PL=0
MOVL C01134 V=800.0 PL=0
MOVL C01135 V=800.0 PL=0
MOVL C01136 V=800.0 PL=0
MOVL C01137 V=800.0 PL=0
MOVL C01138 V=800.0 PL=0
MOVL C01139 V=800.0 PL=0
MOVL C01140 V=800.0 PL=0
MOVL C01141 V=800.0 PL=0
MOVL C01142 V=800.0 PL=0
MOVL C01143 V=800.0 PL=0
MOVL C01144 V=800.0 PL=0
MOVL C01145 V=800.0 PL=0
MOVL C01146 V=800.0 PL=0
MOVL C01147 V=800.0 PL=0
MOVL C01148 V=800.0 PL=0
MOVL C01149 V=800.0 PL=0
MOVL C01150 V=800.0 PL=0
MOVL C01151 V=800.0 PL=0
MOVL C01152 V=800.0 PL=0
MOVL C01153 V=800.0 PL=0
MOVL C01154 V=800.0 PL=0
MOVL C01155 V=800.0 PL=0
MOVL C01156 V=800.0 PL=0
MOVL C01157 V=800.0 PL=0
MOVL C01158 V=800.0 PL=0
MOVL C01159 V=800.0 PL=0
MOVL C01160 V=800.0 PL=0
MOVL C01161 V=800.0 PL=0
MOVL C01162 V=800.0 PL=0
MOVL C01163 V=800.0 PL=0
MOVL C01164 V=800.0 PL=0
MOVL C01165 V=800.0 PL=0
MOVL C01166 V=800.0 PL=0
MOVL C01167 V=800.0 PL=0
MOVL C01168 V=800.0 PL=0
MOVL C01169 V=800.0 PL=0
MOVL C01170 V=800.0 PL=0
MOVL C01171 V=800.0 PL=0
MOVL C01172 V=800.0 PL=0
MOVL C01173 V=800.0 PL=0
MOVL C01174 V=800.0 PL=0
MOVL C01175 V=800.0 PL=0
MOVL C01176 V=800.0 PL=0
MOVL C01177 V=800.0 PL=0
MOVL C01178 V=800.0 PL=0
MOVL C01179 V=800.0 PL=0
MOVL C01180 V=800.0 PL=0
MOVL C01181 V=800.0 PL=0
MOVL C01182 V=800.0 PL=0
MOVL C01183 V=800.0 PL=0
MOVL C01184 V=800.0 PL=0
MOVL C01185 V=800.0 PL=0
MOVL C01186 V=800.0 PL=0
MOVL C01187 V=800.0 PL=0
MOVL C01188 V=800.0 PL=0
MOVL C01189 V=800.0 PL=0
MOVL C01190 V=800.0 PL=0
MOVL C01191 V=800.0 PL=0
MOVL C01192 V=800.0 PL=0
MOVL C01193 V=800.0 PL=0
MOVL C01194 V=800.0 PL=0
MOVL C01195 V=800.0 PL=0
MOVL C01196 V=800.0 PL=0
MOVL C01197 V=800.0 PL=0
MOVL C01198 V=800.0 PL=0
MOVL C01199 V=800.0 PL=0
MOVL C01200 V=800.0 PL=0
MOVL C01201 V=800.0 PL=0
MOVL C01202 V=800.0 PL=0
MOVL C01203 V=800.0 PL=0
MOVL C01204 V=800.0 PL=0
MOVL C01205 V=800.0 PL=0
MOVL C01206 V=800.0 PL=0
MOVL C01207 V=800.0 PL=0
MOVL C01208 V=800.0 PL=0
MOVL C01209 V=800.0 PL=0
MOVL C01210 V=800.0 PL=0
MOVL C01211 V=800.0 PL=0
MOVL C01212 V=800.0 PL=0
MOVL C01213 V=800.0 PL=0
MOVL C01214 V=800.0 PL=0
MOVL C01215 V=800.0 PL=0
MOVL C01216 V=800.0 PL=0
MOVL C01217 V=800.0 PL=0
MOVL C01218 V=800.0 PL=0
MOVL C01219 V=800.0 PL=0
MOVL C01220 V=800.0 PL=0
MOVL C01221 V=800.0 PL=0
MOVL C01222 V=800.0 PL=0
MOVL C01223 V=800.0 PL=0
MOVL C01224 V=800.0 PL=0
MOVL C01225 V=800.0 PL=0
MOVL C01226 V=800.0 PL=0
MOVL C01227 V=800.0 PL=0
MOVL C01228 V=800.0 PL=0
MOVL C01229 V=800.0 PL=0
MOVL C01230 V=800.0 PL=0
MOVL C01231 V=800.0 PL=0
MOVL C01232 V=800.0 PL=0
MOVL C01233 V=800.0 PL=0
MOVL C01234 V=800.0 PL=0
MOVL C01235 V=800.0 PL=0
MOVL C01236 V=800.0 PL=0
MOVL C01237 V=800.0 PL=0
MOVL C01238 V=800.0 PL=0
MOVL C01239 V=800.0 PL=0
MOVL C01240 V=800.0 PL=0
MOVL C01241 V=800.0 PL=0
MOVL C01242 V=800.0 PL=0
MOVL C01243 V=800.0 PL=0
MOVL C01244 V=800.0 PL=0
MOVL C01245 V=800.0 PL=0
MOVL C01246 V=800.0 PL=0
MOVL C01247 V=800.0 PL=0
MOVL C01248 V=800.0 PL=0
MOVL C01249 V=800.0 PL=0
MOVL C01250 V=800.0 PL=0
MOVL C01251 V=800.0 PL=0
MOVL C01252 V=800.0 PL=0
MOVL C01253 V=800.0 PL=0
MOVL C01254 V=800.0 PL=0
MOVL C01255 V=800.0 PL=0
MOVL C01256 V=800.0 PL=0
MOVL C01257 V=800.0 PL=0
MOVL C01258 V=800.0 PL=0
MOVL C01259 V=800.0 PL=0
MOVL C01260 V=800.0 PL=0
MOVL C01261 V=800.0 PL=0
MOVL C01262 V=800.0 PL=0
MOVL C01263 V=800.0 PL=0
MOVL C01264 V=800.0 PL=0
MOVL C01265 V=800.0 PL=0
MOVL C01266 V=800.0 PL=0
MOVL C01267 V=800.0 PL=0
MOVL C01268 V=800.0 PL=0
MOVL C01269 V=800.0 PL=0
MOVL C01270 V=800.0 PL=0
MOVL C01271 V=800.0 PL=0
MOVL C01272 V=800.0 PL=0
MOVL C01273 V=800.0 PL=0
MOVL C01274 V=800.0 PL=0
MOVL C01275 V=800.0 PL=0
MOVL C01276 V=800.0 PL=0
MOVL C01277 V=800.0 PL=0
MOVL C01278 V=800.0 PL=0
MOVL C01279 V=800.0 PL=0
MOVL C01280 V=800.0 PL=0
MOVL C01281 V=800.0 PL=0
MOVL C01282 V=800.0 PL=0
MOVL C01283 V=800.0 PL=0
MOVL C01284 V=800.0 PL=0
MOVL C01285 V=800.0 PL=0
MOVL C01286 V=800.0 PL=0
MOVL C01287 V=800.0 PL=0
MOVL C01288 V=800.0 PL=0
MOVL C01289 V=800.0 PL=0
MOVL C01290 V=800.0 PL=0
MOVL C01291 V=800.0 PL=0
MOVL C01292 V=800.0 PL=0
MOVL C01293 V=800.0 PL=0
MOVL C01294 V=800.0 PL=0
MOVL C01295 V=800.0 PL=0
MOVL C01296 V=800.0 PL=0
MOVL C01297 V=800.0 PL=0
MOVL C01298 V=800.0 PL=0
MOVL C01299 V=800.0 PL=0
MOVL C01300 V=800.0 PL=0
MOVL C01301 V=800.0 PL=0
MOVL C01302 V=800.0 PL=0
MOVL C01303 V=800.0 PL=0
MOVL C01304 V=800.0 PL=0
MOVL C01305 V=800.0 PL=0
MOVL C01306 V=800.0 PL=0
MOVL C01307 V=800.0 PL=0
MOVL C01308 V=800.0 PL=0
MOVL C01309 V=800.0 PL=0
MOVL C01310 V=800.0 PL=0
MOVL C01311 V=800.0 PL=0
MOVL C01312 V=800.0 PL=0
MOVL C01313 V=800.0 PL=0
MOVL C01314 V=800.0 PL=0
MOVL C01315 V=800.0 PL=0
MOVL C01316 V=800.0 PL=0
MOVL C01317 V=800.0 PL=0
MOVL C01318 V=800.0 PL=0
MOVL C01319 V=800.0 PL=0
MOVL C01320 V=800.0 PL=0
MOVL C01321 V=800.0 PL=0
MOVL C01322 V=800.0 PL=0
MOVL C01323 V=800.0 PL=0
MOVL C01324 V=800.0 PL=0
MOVL C01325 V=800.0 PL=0
MOVL C01326 V=800.0 PL=0
MOVL C01327 V=800.0 PL=0
MOVL C01328 V=800.0 PL=0
MOVL C01329 V=800.0 PL=0
MOVL C01330 V=800.0 PL=0
MOVL C01331 V=800.0 PL=0
MOVL C01332 V=800.0 PL=0
MOVL C01333 V=800.0 PL=0
MOVL C01334 V=800.0 PL=0
MOVL C01335 V=800.0 PL=0
MOVL C01336 V=800.0 PL=0
MOVL C01337 V=800.0 PL=0
MOVL C01338 V=800.0 PL=0
MOVL C01339 V=800.0 PL=0
MOVL C01340 V=800.0 PL=0
MOVL C01341 V=800.0 PL=0
MOVL C01342 V=800.0 PL=0
MOVL C01343 V=800.0 PL=0
MOVL C01344 V=800.0 PL=0
MOVL C01345 V=800.0 PL=0
MOVL C01346 V=800.0 PL=0
MOVL C01347 V=800.0 PL=0
MOVL C01348 V=800.0 PL=0
MOVL C01349 V=800.0 PL=0
MOVL C01350 V=800.0 PL=0
MOVL C01351 V=800.0 PL=0
MOVL C01352 V=800.0 PL=0
MOVL C01353 V=800.0 PL=0
MOVL C01354 V=800.0 PL=0
MOVL C01355 V=800.0 PL=0
MOVL C01356 V=800.0 PL=0
MOVL C01357 V=800.0 PL=0
MOVL C01358 V=800.0 PL=0
MOVL C01359 V=800.0 PL=0
MOVL C01360 V=800.0 PL=0
MOVL C01361 V=800.0 PL=0
MOVL C01362 V=800.0 PL=0
MOVL C01363 V=800.0 PL=0
MOVL C01364 V=800.0 PL=0
MOVL C01365 V=800.0 PL=0
MOVL C01366 V=800.0 PL=0
MOVL C01367 V=800.0 PL=0
MOVL C01368 V=800.0 PL=0
MOVL C01369 V=800.0 PL=0
MOVL C01370 V=800.0 PL=0
MOVL C01371 V=800.0 PL=0
MOVL C01372 V=800.0 PL=0
MOVL C01373 V=800.0 PL=0
MOVL C01374 V=800.0 PL=0
MOVL C01375 V=800.0 PL=0
MOVL C01376 V=800.0 PL=0
MOVL C01377 V=800.0 PL=0
MOVL C01378 V=800.0 PL=0
MOVL C01379 V=800.0 PL=0
MOVL C01380 V=800.0 PL=0
MOVL C01381 V=800.0 PL=0
MOVL C01382 V=800.0 PL=0
MOVL C01383 V=800.0 PL=0
MOVL C01384 V=800.0 PL=0
MOVL C01385 V=800.0 PL=0
MOVL C01386 V=800.0 PL=0
MOVL C01387 V=800.0 PL=0
MOVL C01388 V=800.0 PL=0
MOVL C01389 V=800.0 PL=0
MOVL C01390 V=800.0 PL=0
MOVL C01391 V=800.0 PL=0
MOVL C01392 V=800.0 PL=0
MOVL C01393 V=800.0 PL=0
MOVL C01394 V=800.0 PL=0
MOVL C01395 V=800.0 PL=0
MOVL C01396 V=800.0 PL=0
MOVL C01397 V=800.0 PL=0
MOVL C01398 V=800.0 PL=0
MOVL C01399 V=800.0 PL=0
MOVL C01400 V=800.0 PL=0
MOVL C01401 V=800.0 PL=0
MOVL C01402 V=800.0 PL=0
MOVL C01403 V=800.0 PL=0
MOVL C01404 V=800.0 PL=0
MOVL C01405 V=800.0 PL=0
MOVL C01406 V=800.0 PL=0
MOVL C01407 V=800.0 PL=0
MOVL C01408 V=800.0 PL=0
MOVL C01409 V=800.0 PL=0
MOVL C01410 V=800.0 PL=0
MOVL C01411 V=800.0 PL=0
MOVL C01412 V=800.0 PL=0
MOVL C01413 V=800.0 PL=0
MOVL C01414 V=800.0 PL=0
MOVL C01415 V=800.0 PL=0
MOVL C01416 V=800.0 PL=0
MOVL C01417 V=800.0 PL=0
MOVL C01418 V=800.0 PL=0
MOVL C01419 V=800.0 PL=0
MOVL C01420 V=800.0 PL=0
MOVL C01421 V=800.0 PL=0
MOVL C01422 V=800.0 PL=0
MOVL C01423 V=800.0 PL=0
MOVL C01424 V=800.0 PL=0
MOVL C01425 V=800.0 PL=0
MOVL C01426 V=800.0 PL=0
MOVL C01427 V=800.0 PL=0
MOVL C01428 V=800.0 PL=0
MOVL C01429 V=800.0 PL=0
MOVL C01430 V=800.0 PL=0
MOVL C01431 V=800.0 PL=0
MOVL C01432 V=800.0 PL=0
MOVL C01433 V=800.0 PL=0
MOVL C01434 V=800.0 PL=0
MOVL C01435 V=800.0 PL=0
MOVL C01436 V=800.0 PL=0
MOVL C01437 V=800.0 PL=0
MOVL C01438 V=800.0 PL=0
MOVL C01439 V=800.0 PL=0
MOVL C01440 V=800.0 PL=0
MOVL C01441 V=800.0 PL=0
MOVL C01442 V=800.0 PL=0
MOVL C01443 V=800.0 PL=0
MOVL C01444 V=800.0 PL=0
MOVL C01445 V=800.0 PL=0
MOVL C01446 V=800.0 PL=0
MOVL C01447 V=800.0 PL=0
MOVL C01448 V=800.0 PL=0
MOVL C01449 V=800.0 PL=0
MOVL C01450 V=800.0 PL=0
MOVL C01451 V=800.0 PL=0
MOVL C01452 V=800.0 PL=0
MOVL C01453 V=800.0 PL=0
MOVL C01454 V=800.0 PL=0
MOVL C01455 V=800.0 PL=0
MOVL C01456 V=800.0 PL=0
MOVL C01457 V=800.0 PL=0
MOVL C01458 V=800.0 PL=0
MOVL C01459 V=800.0 PL=0
MOVL C01460 V=800.0 PL=0
MOVL C01461 V=800.0 PL=0
MOVL C01462 V=800.0 PL=0
MOVL C01463 V=800.0 PL=0
MOVL C01464 V=800.0 PL=0
MOVL C01465 V=800.0 PL=0
MOVL C01466 V=800.0 PL=0
MOVL C01467 V=800.0 PL=0
MOVL C01468 V=800.0 PL=0
MOVL C01469 V=800.0 PL=0
MOVL C01470 V=800.0 PL=0
MOVL C01471 V=800.0 PL=0
MOVL C01472 V=800.0 PL=0
MOVL C01473 V=800.0 PL=0
MOVL C01474 V=800.0 PL=0
MOVL C01475 V=800.0 PL=0
MOVL C01476 V=800.0 PL=0
MOVL C01477 V=800.0 PL=0
MOVL C01478 V=800.0 PL=0
MOVL C01479 V=800.0 PL=0
MOVL C01480 V=800.0 PL=0
MOVL C01481 V=800.0 PL=0
MOVL C01482 V=800.0 PL=0
MOVL C01483 V=800.0 PL=0
MOVL C01484 V=800.0 PL=0
MOVL C01485 V=800.0 PL=0
MOVL C01486 V=800.0 PL=0
MOVL C01487 V=800.0 PL=0
MOVL C01488 V=800.0 PL=0
MOVL C01489 V=800.0 PL=0
MOVL C01490 V=800.0 PL=0
MOVL C01491 V=800.0 PL=0
MOVL C01492 V=800.0 PL=0
MOVL C01493 V=800.0 PL=0
MOVL C01494 V=800.0 PL=0
MOVL C01495 V=800.0 PL=0
MOVL C01496 V=800.0 PL=0
MOVL C01497 V=800.0 PL=0
MOVL C01498 V=800.0 PL=0
MOVL C01499 V=800.0 PL=0
MOVL C01500 V=800.0 PL=0
MOVL C01501 V=800.0 PL=0
MOVL C01502 V=800.0 PL=0
MOVL C01503 V=800.0 PL=0
MOVL C01504 V=800.0 PL=0
MOVL C01505 V=800.0 PL=0
MOVL C01506 V=800.0 PL=0
MOVL C01507 V=800.0 PL=0
MOVL C01508 V=800.0 PL=0
MOVL C01509 V=800.0 PL=0
MOVL C01510 V=800.0 PL=0
MOVL C01511 V=800.0 PL=0
MOVL C01512 V=800.0 PL=0
MOVL C01513 V=800.0 PL=0
MOVL C01514 V=800.0 PL=0
MOVL C01515 V=800.0 PL=0
MOVL C01516 V=800.0 PL=0
MOVL C01517 V=800.0 PL=0
MOVL C01518 V=800.0 PL=0
MOVL C01519 V=800.0 PL=0
MOVL C01520 V=800.0 PL=0
MOVL C01521 V=800.0 PL=0
MOVL C01522 V=800.0 PL=0
MOVL C01523 V=800.0 PL=0
MOVL C01524 V=800.0 PL=0
MOVL C01525 V=800.0 PL=0
MOVL C01526 V=800.0 PL=0
MOVL C01527 V=800.0 PL=0
MOVL C01528 V=800.0 PL=0
MOVL C01529 V=800.0 PL=0
MOVL C01530 V=800.0 PL=0
MOVL C01531 V=800.0 PL=0
MOVL C01532 V=800.0 PL=0
MOVL C01533 V=800.0 PL=0
MOVL C01534 V=800.0 PL=0
MOVL C01535 V=800.0 PL=0
MOVL C01536 V=800.0 PL=0
MOVL C01537 V=800.0 PL=0
MOVL C01538 V=800.0 PL=0
MOVL C01539 V=800.0 PL=0
MOVL C01540 V=800.0 PL=0
MOVL C01541 V=800.0 PL=0
MOVL C01542 V=800.0 PL=0
MOVL C01543 V=800.0 PL=0
MOVL C01544 V=800.0 PL=0
MOVL C01545 V=800.0 PL=0
MOVL C01546 V=800.0 PL=0
MOVL C01547 V=800.0 PL=0
MOVL C01548 V=800.0 PL=0
MOVL C01549 V=800.0 PL=0
MOVL C01550 V=800.0 PL=0
MOVL C01551 V=800.0 PL=0
MOVL C01552 V=800.0 PL=0
MOVL C01553 V=800.0 PL=0
MOVL C01554 V=800.0 PL=0
MOVL C01555 V=800.0 PL=0
MOVL C01556 V=800.0 PL=0
MOVL C01557 V=800.0 PL=0
MOVL C01558 V=800.0 PL=0
MOVL C01559 V=800.0 PL=0
MOVL C01560 V=800.0 PL=0
MOVL C01561 V=800.0 PL=0
MOVL C01562 V=800.0 PL=0
MOVL C01563 V=800.0 PL=0
MOVL C01564 V=800.0 PL=0
MOVL C01565 V=800.0 PL=0
MOVL C01566 V=800.0 PL=0
MOVL C01567 V=800.0 PL=0
MOVL C01568 V=800.0 PL=0
MOVL C01569 V=800.0 PL=0
MOVL C01570 V=800.0 PL=0
MOVL C01571 V=800.0 PL=0
MOVL C01572 V=800.0 PL=0
MOVL C01573 V=800.0 PL=0
MOVL C01574 V=800.0 PL=0
MOVL C01575 V=800.0 PL=0
MOVL C01576 V=800.0 PL=0
MOVL C01577 V=800.0 PL=0
MOVL C01578 V=800.0 PL=0
MOVL C01579 V=800.0 PL=0
MOVL C01580 V=800.0 PL=0
MOVL C01581 V=800.0 PL=0
MOVL C01582 V=800.0 PL=0
MOVL C01583 V=800.0 PL=0
MOVL C01584 V=800.0 PL=0
MOVL C01585 V=800.0 PL=0
MOVL C01586 V=800.0 PL=0
MOVL C01587 V=800.0 PL=0
MOVL C01588 V=800.0 PL=0
MOVL C01589 V=800.0 PL=0
MOVL C01590 V=800.0 PL=0
MOVL C01591 V=800.0 PL=0
MOVL C01592 V=800.0 PL=0
MOVL C01593 V=800.0 PL=0
MOVL C01594 V=800.0 PL=0
MOVL C01595 V=800.0 PL=0
MOVL C01596 V=800.0 PL=0
MOVL C01597 V=800.0 PL=0
MOVL C01598 V=800.0 PL=0
MOVL C01599 V=800.0 PL=0
MOVL C01600 V=800.0 PL=0
MOVL C01601 V=800.0 PL=0
MOVL C01602 V=800.0 PL=0
MOVL C01603 V=800.0 PL=0
MOVL C01604 V=800.0 PL=0
MOVL C01605 V=800.0 PL=0
MOVL C01606 V=800.0 PL=0
MOVL C01607 V=800.0 PL=0
MOVL C01608 V=800.0 PL=0
MOVL C01609 V=800.0 PL=0
MOVL C01610 V=800.0 PL=0
MOVL C01611 V=800.0 PL=0
MOVL C01612 V=800.0 PL=0
MOVL C01613 V=800.0 PL=0
MOVL C01614 V=800.0 PL=0
MOVL C01615 V=800.0 PL=0
MOVL C01616 V=800.0 PL=0
MOVL C01617 V=800.0 PL=0
MOVL C01618 V=800.0 PL=0
MOVL C01619 V=800.0 PL=0
MOVL C01620 V=800.0 PL=0
MOVL C01621 V=800.0 PL=0
MOVL C01622 V=800.0 PL=0
MOVL C01623 V=800.0 PL=0
MOVL C01624 V=800.0 PL=0
MOVL C01625 V=800.0 PL=0
MOVL C01626 V=800.0 PL=0
MOVL C01627 V=800.0 PL=0
MOVL C01628 V=800.0 PL=0
MOVL C01629 V=800.0 PL=0
MOVL C01630 V=800.0 PL=0
MOVL C01631 V=800.0 PL=0
MOVL C01632 V=800.0 PL=0
MOVL C01633 V=800.0 PL=0
MOVL C01634 V=800.0 PL=0
MOVL C01635 V=800.0 PL=0
MOVL C01636 V=800.0 PL=0
MOVL C01637 V=800.0 PL=0
MOVL C01638 V=800.0 PL=0
MOVL C01639 V=800.0 PL=0
MOVL C01640 V=800.0 PL=0
MOVL C01641 V=800.0 PL=0
MOVL C01642 V=800.0 PL=0
MOVL C01643 V=800.0 PL=0
MOVL C01644 V=800.0 PL=0
MOVL C01645 V=800.0 PL=0
MOVL C01646 V=800.0 PL=0
MOVL C01647 V=800.0 PL=0
MOVL C01648 V=800.0 PL=0
MOVL C01649 V=800.0 PL=0
MOVL C01650 V=800.0 PL=0
MOVL C01651 V=800.0 PL=0
MOVL C01652 V=800.0 PL=0
MOVL C01653 V=800.0 PL=0
MOVL C01654 V=800.0 PL=0
MOVL C01655 V=800.0 PL=0
MOVL C01656 V=800.0 PL=0
MOVL C01657 V=800.0 PL=0
MOVL C01658 V=800.0 PL=0
MOVL C01659 V=800.0 PL=0
MOVL C01660 V=800.0 PL=0
MOVL C01661 V=800.0 PL=0
MOVL C01662 V=800.0 PL=0
MOVL C01663 V=800.0 PL=0
MOVL C01664 V=800.0 PL=0
MOVL C01665 V=800.0 PL=0
MOVL C01666 V=800.0 PL=0
MOVL C01667 V=800.0 PL=0
MOVL C01668 V=800.0 PL=0
MOVL C01669 V=800.0 PL=0
MOVL C01670 V=800.0 PL=0
MOVL C01671 V=800.0 PL=0
MOVL C01672 V=800.0 PL=0
MOVL C01673 V=800.0 PL=0
MOVL C01674 V=800.0 PL=0
MOVL C01675 V=800.0 PL=0
MOVL C01676 V=800.0 PL=0
MOVL C01677 V=800.0 PL=0
MOVL C01678 V=800.0 PL=0
MOVL C01679 V=800.0 PL=0
MOVL C01680 V=800.0 PL=0
MOVL C01681 V=800.0 PL=0
MOVL C01682 V=800.0 PL=0
MOVL C01683 V=800.0 PL=0
MOVL C01684 V=800.0 PL=0
MOVL C01685 V=800.0 PL=0
MOVL C01686 V=800.0 PL=0
MOVL C01687 V=800.0 PL=0
MOVL C01688 V=800.0 PL=0
MOVL C01689 V=800.0 PL=0
MOVL C01690 V=800.0 PL=0
MOVL C01691 V=800.0 PL=0
MOVL C01692 V=800.0 PL=0
MOVL C01693 V=800.0 PL=0
MOVL C01694 V=800.0 PL=0
MOVL C01695 V=800.0 PL=0
MOVL C01696 V=800.0 PL=0
MOVL C01697 V=800.0 PL=0
MOVL C01698 V=800.0 PL=0
MOVL C01699 V=800.0 PL=0
MOVL C01700 V=800.0 PL=0
MOVL C01701 V=800.0 PL=0
MOVL C01702 V=800.0 PL=0
MOVL C01703 V=800.0 PL=0
MOVL C01704 V=800.0 PL=0
MOVL C01705 V=800.0 PL=0
MOVL C01706 V=800.0 PL=0
MOVL C01707 V=800.0 PL=0
MOVL C01708 V=800.0 PL=0
MOVL C01709 V=800.0 PL=0
MOVL C01710 V=800.0 PL=0
MOVL C01711 V=800.0 PL=0
MOVL C01712 V=800.0 PL=0
MOVL C01713 V=800.0 PL=0
MOVL C01714 V=800.0 PL=0
MOVL C01715 V=800.0 PL=0
MOVL C01716 V=800.0 PL=0
MOVL C01717 V=800.0 PL=0
MOVL C01718 V=800.0 PL=0
MOVL C01719 V=800.0 PL=0
MOVL C01720 V=800.0 PL=0
MOVL C01721 V=800.0 PL=0
MOVL C01722 V=800.0 PL=0
MOVL C01723 V=800.0 PL=0
MOVL C01724 V=800.0 PL=0
MOVL C01725 V=800.0 PL=0
MOVL C01726 V=800.0 PL=0
MOVL C01727 V=800.0 PL=0
MOVL C01728 V=800.0 PL=0
MOVL C01729 V=800.0 PL=0
MOVL C01730 V=800.0 PL=0
MOVL C01731 V=800.0 PL=0
MOVL C01732 V=800.0 PL=0
MOVL C01733 V=800.0 PL=0
MOVL C01734 V=800.0 PL=0
MOVL C01735 V=800.0 PL=0
MOVL C01736 V=800.0 PL=0
MOVL C01737 V=800.0 PL=0
MOVL C01738 V=800.0 PL=0
MOVL C01739 V=800.0 PL=0
MOVL C01740 V=800.0 PL=0
MOVL C01741 V=800.0 PL=0
MOVL C01742 V=800.0 PL=0
MOVL C01743 V=800.0 PL=0
MOVL C01744 V=800.0 PL=0
MOVL C01745 V=800.0 PL=0
MOVL C01746 V=800.0 PL=0
MOVL C01747 V=800.0 PL=0
MOVL C01748 V=800.0 PL=0
MOVL C01749 V=800.0 PL=0
MOVL C01750 V=800.0 PL=0
MOVL C01751 V=800.0 PL=0
MOVL C01752 V=800.0 PL=0
MOVL C01753 V=800.0 PL=0
MOVL C01754 V=800.0 PL=0
MOVL C01755 V=800.0 PL=0
MOVL C01756 V=800.0 PL=0
MOVL C01757 V=800.0 PL=0
MOVL C01758 V=800.0 PL=0
MOVL C01759 V=800.0 PL=0
MOVL C01760 V=800.0 PL=0
MOVL C01761 V=800.0 PL=0
MOVL C01762 V=800.0 PL=0
MOVL C01763 V=800.0 PL=0
MOVL C01764 V=800.0 PL=0
MOVL C01765 V=800.0 PL=0
MOVL C01766 V=800.0 PL=0
MOVL C01767 V=800.0 PL=0
MOVL C01768 V=800.0 PL=0
MOVL C01769 V=800.0 PL=0
MOVL C01770 V=800.0 PL=0
MOVL C01771 V=800.0 PL=0
MOVL C01772 V=800.0 PL=0
MOVL C01773 V=800.0 PL=0
MOVL C01774 V=800.0 PL=0
MOVL C01775 V=800.0 PL=0
MOVL C01776 V=800.0 PL=0
MOVL C01777 V=800.0 PL=0
MOVL C01778 V=800.0 PL=0
MOVL C01779 V=800.0 PL=0
MOVL C01780 V=800.0 PL=0
MOVL C01781 V=800.0 PL=0
MOVL C01782 V=800.0 PL=0
MOVL C01783 V=800.0 PL=0
MOVL C01784 V=800.0 PL=0
MOVL C01785 V=800.0 PL=0
MOVL C01786 V=800.0 PL=0
MOVL C01787 V=800.0 PL=0
MOVL C01788 V=800.0 PL=0
MOVL C01789 V=800.0 PL=0
MOVL C01790 V=800.0 PL=0
MOVL C01791 V=800.0 PL=0
MOVL C01792 V=800.0 PL=0
MOVL C01793 V=800.0 PL=0
MOVL C01794 V=800.0 PL=0
MOVL C01795 V=800.0 PL=0
MOVL C01796 V=800.0 PL=0
MOVL C01797 V=800.0 PL=0
MOVL C01798 V=800.0 PL=0
MOVL C01799 V=800.0 PL=0
MOVL C01800 V=800.0 PL=0
MOVL C01801 V=800.0 PL=0
MOVL C01802 V=800.0 PL=0
MOVL C01803 V=800.0 PL=0
MOVL C01804 V=800.0 PL=0
MOVL C01805 V=800.0 PL=0
MOVL C01806 V=800.0 PL=0
MOVL C01807 V=800.0 PL=0
MOVL C01808 V=800.0 PL=0
MOVL C01809 V=800.0 PL=0
MOVL C01810 V=800.0 PL=0
MOVL C01811 V=800.0 PL=0
MOVL C01812 V=800.0 PL=0
MOVL C01813 V=800.0 PL=0
MOVL C01814 V=800.0 PL=0
MOVL C01815 V=800.0 PL=0
MOVL C01816 V=800.0 PL=0
MOVL C01817 V=800.0 PL=0
MOVL C01818 V=800.0 PL=0
MOVL C01819 V=800.0 PL=0
MOVL C01820 V=800.0 PL=0
MOVL C01821 V=800.0 PL=0
MOVL C01822 V=800.0 PL=0
MOVL C01823 V=800.0 PL=0
MOVL C01824 V=800.0 PL=0
MOVL C01825 V=800.0 PL=0
MOVL C01826 V=800.0 PL=0
MOVL C01827 V=800.0 PL=0
MOVL C01828 V=800.0 PL=0
MOVL C01829 V=800.0 PL=0
MOVL C01830 V=800.0 PL=0
MOVL C01831 V=800.0 PL=0
MOVL C01832 V=800.0 PL=0
MOVL C01833 V=800.0 PL=0
MOVL C01834 V=800.0 PL=0
MOVL C01835 V=800.0 PL=0
MOVL C01836 V=800.0 PL=0
MOVL C01837 V=800.0 PL=0
MOVL C01838 V=800.0 PL=0
MOVL C01839 V=800.0 PL=0
MOVL C01840 V=800.0 PL=0
MOVL C01841 V=800.0 PL=0
MOVL C01842 V=800.0 PL=0
MOVL C01843 V=800.0 PL=0
MOVL C01844 V=800.0 PL=0
MOVL C01845 V=800.0 PL=0
MOVL C01846 V=800.0 PL=0
MOVL C01847 V=800.0 PL=0
MOVL C01848 V=800.0 PL=0
MOVL C01849 V=800.0 PL=0
MOVL C01850 V=800.0 PL=0
MOVL C01851 V=800.0 PL=0
MOVL C01852 V=800.0 PL=0
MOVL C01853 V=800.0 PL=0
MOVL C01854 V=800.0 PL=0
MOVL C01855 V=800.0 PL=0
MOVL C01856 V=800.0 PL=0
MOVL C01857 V=800.0 PL=0
MOVL C01858 V=800.0 PL=0
MOVL C01859 V=800.0 PL=0
MOVL C01860 V=800.0 PL=0
MOVL C01861 V=800.0 PL=0
MOVL C01862 V=800.0 PL=0
MOVL C01863 V=800.0 PL=0
MOVL C01864 V=800.0 PL=0
MOVL C01865 V=800.0 PL=0
MOVL C01866 V=800.0 PL=0
MOVL C01867 V=800.0 PL=0
MOVL C01868 V=800.0 PL=0
MOVL C01869 V=800.0 PL=0
MOVL C01870 V=800.0 PL=0
MOVL C01871 V=800.0 PL=0
MOVL C01872 V=800.0 PL=0
MOVL C01873 V=800.0 PL=0
MOVL C01874 V=800.0 PL=0
MOVL C01875 V=800.0 PL=0
MOVL C01876 V=800.0 PL=0
MOVL C01877 V=800.0 PL=0
MOVL C01878 V=800.0 PL=0
MOVL C01879 V=800.0 PL=0
MOVL C01880 V=800.0 PL=0
MOVL C01881 V=800.0 PL=0
MOVL C01882 V=800.0 PL=0
MOVL C01883 V=800.0 PL=0
MOVL C01884 V=800.0 PL=0
MOVL C01885 V=800.0 PL=0
MOVL C01886 V=800.0 PL=0
MOVL C01887 V=800.0 PL=0
MOVL C01888 V=800.0 PL=0
MOVL C01889 V=800.0 PL=0
MOVL C01890 V=800.0 PL=0
MOVL C01891 V=800.0 PL=0
MOVL C01892 V=800.0 PL=0
MOVL C01893 V=800.0 PL=0
MOVL C01894 V=800.0 PL=0
MOVL C01895 V=800.0 PL=0
MOVL C01896 V=800.0 PL=0
MOVL C01897 V=800.0 PL=0
MOVL C01898 V=800.0 PL=0
MOVL C01899 V=800.0 PL=0
MOVL C01900 V=800.0 PL=0
MOVL C01901 V=800.0 PL=0
MOVL C01902 V=800.0 PL=0
MOVL C01903 V=800.0 PL=0
MOVL C01904 V=800.0 PL=0
MOVL C01905 V=800.0 PL=0
MOVL C01906 V=800.0 PL=0
MOVL C01907 V=800.0 PL=0
MOVL C01908 V=800.0 PL=0
MOVL C01909 V=800.0 PL=0
MOVL C01910 V=800.0 PL=0
MOVL C01911 V=800.0 PL=0
MOVL C01912 V=800.0 PL=0
MOVL C01913 V=800.0 PL=0
MOVL C01914 V=800.0 PL=0
MOVL C01915 V=800.0 PL=0
MOVL C01916 V=800.0 PL=0
MOVL C01917 V=800.0 PL=0
MOVL C01918 V=800.0 PL=0
MOVL C01919 V=800.0 PL=0
MOVL C01920 V=800.0 PL=0
MOVL C01921 V=800.0 PL=0
MOVL C01922 V=800.0 PL=0
MOVL C01923 V=800.0 PL=0
MOVL C01924 V=800.0 PL=0
MOVL C01925 V=800.0 PL=0
MOVL C01926 V=800.0 PL=0
MOVL C01927 V=800.0 PL=0
MOVL C01928 V=800.0 PL=0
MOVL C01929 V=800.0 PL=0
MOVL C01930 V=800.0 PL=0
MOVL C01931 V=800.0 PL=0
MOVL C01932 V=800.0 PL=0
MOVL C01933 V=800.0 PL=0
MOVL C01934 V=800.0 PL=0
MOVL C01935 V=800.0 PL=0
MOVL C01936 V=800.0 PL=0
MOVL C01937 V=800.0 PL=0
MOVL C01938 V=800.0 PL=0
MOVL C01939 V=800.0 PL=0
MOVL C01940 V=800.0 PL=0
MOVL C01941 V=800.0 PL=0
MOVL C01942 V=800.0 PL=0
MOVL C01943 V=800.0 PL=0
MOVL C01944 V=800.0 PL=0
MOVL C01945 V=800.0 PL=0
MOVL C01946 V=800.0 PL=0
MOVL C01947 V=800.0 PL=0
MOVL C01948 V=800.0 PL=0
MOVL C01949 V=800.0 PL=0
MOVL C01950 V=800.0 PL=0
MOVL C01951 V=800.0 PL=0
MOVL C01952 V=800.0 PL=0
MOVL C01953 V=800.0 PL=0
MOVL C01954 V=800.0 PL=0
MOVL C01955 V=800.0 PL=0
MOVL C01956 V=800.0 PL=0
MOVL C01957 V=800.0 PL=0
MOVL C01958 V=800.0 PL=0
MOVL C01959 V=800.0 PL=0
MOVL C01960 V=800.0 PL=0
MOVL C01961 V=800.0 PL=0
MOVL C01962 V=800.0 PL=0
MOVL C01963 V=800.0 PL=0
MOVL C01964 V=800.0 PL=0
MOVL C01965 V=800.0 PL=0
MOVL C01966 V=800.0 PL=0
MOVL C01967 V=800.0 PL=0
MOVL C01968 V=800.0 PL=0
MOVL C01969 V=800.0 PL=0
MOVL C01970 V=800.0 PL=0
MOVL C01971 V=800.0 PL=0
MOVL C01972 V=800.0 PL=0
MOVL C01973 V=800.0 PL=0
MOVL C01974 V=800.0 PL=0
MOVL C01975 V=800.0 PL=0
MOVL C01976 V=800.0 PL=0
MOVL C01977 V=800.0 PL=0
MOVL C01978 V=800.0 PL=0
MOVL C01979 V=800.0 PL=0
MOVL C01980 V=800.0 PL=0
MOVL C01981 V=800.0 PL=0
MOVL C01982 V=800.0 PL=0
MOVL C01983 V=800.0 PL=0
MOVL C01984 V=800.0 PL=0
MOVL C01985 V=800.0 PL=0
MOVL C01986 V=800.0 PL=0
MOVL C01987 V=800.0 PL=0
MOVL C01988 V=800.0 PL=0
MOVL C01989 V=800.0 PL=0
MOVL C01990 V=800.0 PL=0
MOVL C01991 V=800.0 PL=0
MOVL C01992 V=800.0 PL=0
MOVL C01993 V=800.0 PL=0
MOVL C01994 V=800.0 PL=0
MOVL C01995 V=800.0 PL=0
